LIN {X 0,Y 266.137,Z 368.245,A -85,B 0,C 180,E1 -18633.74,E2 -18633.74} C_VEL
LIN {X 0,Y 268.188,Z 298.553,A -85,B 0,C 180,E1 -18635.636,E2 -18635.636} C_VEL
LIN {X 0,Y 265.756,Z 283.808,A -85,B 0,C 180,E1 -18636.272,E2 -18636.272} C_VEL
LIN {X 0,Y 257.715,Z 261.033,A -85,B 0,C 180,E1 -18637.734,E2 -18637.734} C_VEL
LIN {X 0,Y 256.638,Z 256.402,A -85,B 0,C 180,E1 -18639.459,E2 -18639.459} C_VEL
LIN {X 0,Y 256.319,Z 255.078,A -85,B 0,C 180,E1 -18640.158,E2 -18640.158} C_VEL
LIN {X 0,Y 256.217,Z 255.067,A -85,B 0,C 180,E1 -18644.295,E2 -18644.295} C_VEL
LIN {X 0,Y 256.169,Z 255.06,A -85,B 0,C 180,E1 -18647.567,E2 -18647.567} C_VEL
LIN {X 0,Y 256.112,Z 255.08,A -85,B 0,C 180,E1 -18651.116,E2 -18651.116} C_VEL
LIN {X 0,Y 256.058,Z 255.088,A -85,B 0,C 180,E1 -18655.095,E2 -18655.095} C_VEL
LIN {X 0,Y 256.055,Z 255.092,A -85,B 0,C 180,E1 -18658.578,E2 -18658.578} C_VEL
LIN {X 0,Y 256.047,Z 255.086,A -85,B 0,C 180,E1 -18661.707,E2 -18661.707} C_VEL
LIN {X 0,Y 256.054,Z 255.088,A -85,B 0,C 180,E1 -18665.2,E2 -18665.2} C_VEL
LIN {X 0,Y 256.042,Z 255.078,A -85,B 0,C 180,E1 -18669.15,E2 -18669.15} C_VEL
LIN {X 0,Y 256.002,Z 255.095,A -85,B 0,C 180,E1 -18673.343,E2 -18673.343} C_VEL
LIN {X 0,Y 256.017,Z 255.082,A -85,B 0,C 180,E1 -18677.836,E2 -18677.836} C_VEL
LIN {X 0,Y 256.05,Z 255.079,A -85,B 0,C 180,E1 -18680.864,E2 -18680.864} C_VEL
LIN {X 0,Y 256.067,Z 255.089,A -85,B 0,C 180,E1 -18684.814,E2 -18684.814} C_VEL
LIN {X 0,Y 256.067,Z 255.075,A -85,B 0,C 180,E1 -18688.577,E2 -18688.577} C_VEL
LIN {X 0,Y 256.069,Z 255.074,A -85,B 0,C 180,E1 -18692.196,E2 -18692.196} C_VEL
LIN {X 0,Y 256.079,Z 255.087,A -85,B 0,C 180,E1 -18695.698,E2 -18695.698} C_VEL
LIN {X 0,Y 256.118,Z 255.079,A -85,B 0,C 180,E1 -18699.108,E2 -18699.108} C_VEL
LIN {X 0,Y 256.23,Z 255.045,A -85,B 0,C 180,E1 -18704.088,E2 -18704.088} C_VEL
LIN {X 0,Y 256.288,Z 255.053,A -85,B 0,C 180,E1 -18707.334,E2 -18707.334} C_VEL
LIN {X 0,Y 256.438,Z 255.039,A -85,B 0,C 180,E1 -18710.629,E2 -18710.629} C_VEL
LIN {X 0,Y 256.458,Z 255.029,A -85,B 0,C 180,E1 -18713.713,E2 -18713.713} C_VEL
LIN {X 0,Y 256.703,Z 254.992,A -85,B 0,C 180,E1 -18718.437,E2 -18718.437} C_VEL
LIN {X 0,Y 256.706,Z 255.004,A -85,B 0,C 180,E1 -18721.575,E2 -18721.575} C_VEL
LIN {X 0,Y 256.333,Z 255.048,A -85,B 0,C 180,E1 -18725.241,E2 -18725.241} C_VEL
LIN {X 0,Y 256.073,Z 255.082,A -85,B 0,C 180,E1 -18726.119,E2 -18726.119} C_VEL
LIN {X 0,Y 254.757,Z 255.238,A -85,B 0,C 180,E1 -18727.415,E2 -18727.415} C_VEL
LIN {X 0,Y 250.37,Z 255.78,A -85,B 0,C 180,E1 -18730.434,E2 -18730.434} C_VEL
LIN {X 0,Y 249.286,Z 255.921,A -85,B 0,C 180,E1 -18731.786,E2 -18731.786} C_VEL
LIN {X 0,Y 249.193,Z 255.934,A -85,B 0,C 180,E1 -18732.245,E2 -18732.245} C_VEL
LIN {X 0,Y 249.189,Z 255.946,A -85,B 0,C 180,E1 -18736.473,E2 -18736.473} C_VEL
LIN {X 0,Y 249.062,Z 255.947,A -85,B 0,C 180,E1 -18741.526,E2 -18741.526} C_VEL
LIN {X 0,Y 249.102,Z 255.955,A -85,B 0,C 180,E1 -18745.463,E2 -18745.463} C_VEL
LIN {X 0,Y 249.053,Z 255.949,A -85,B 0,C 180,E1 -18748.976,E2 -18748.976} C_VEL
LIN {X 0,Y 249.046,Z 255.96,A -85,B 0,C 180,E1 -18752.429,E2 -18752.429} C_VEL
LIN {X 0,Y 249.03,Z 255.954,A -85,B 0,C 180,E1 -18756.352,E2 -18756.352} C_VEL
LIN {X 0,Y 248.991,Z 255.968,A -85,B 0,C 180,E1 -18760.487,E2 -18760.487} C_VEL
LIN {X 0,Y 248.982,Z 255.97,A -85,B 0,C 180,E1 -18764.891,E2 -18764.891} C_VEL
LIN {X 0,Y 248.999,Z 255.963,A -85,B 0,C 180,E1 -18767.356,E2 -18767.356} C_VEL
LIN {X 0,Y 249.064,Z 255.951,A -85,B 0,C 180,E1 -18772.202,E2 -18772.202} C_VEL
LIN {X 0,Y 249.119,Z 256.035,A -85,B 0,C 180,E1 -18776.259,E2 -18776.259} C_VEL
LIN {X 0,Y 250.073,Z 260.614,A -85,B 0,C 180,E1 -18778.198,E2 -18778.198} C_VEL
LIN {X 0,Y 251.47,Z 267.192,A -85,B 0,C 180,E1 -18780.671,E2 -18780.671} C_VEL
LIN {X 0,Y 257.562,Z 284.54,A -85,B 0,C 180,E1 -18781.846,E2 -18781.846} C_VEL
LIN {X 0,Y 261.408,Z 311.936,A -85,B 0,C 180,E1 -18783.017,E2 -18783.017} C_VEL
LIN {X 0,Y 259.429,Z 375.405,A -85,B 0,C 180,E1 -18784.795,E2 -18784.795} C_VEL
LIN {X 0,Y 258.511,Z 388.458,A -85,B 0,C 180,E1 -18785.45,E2 -18785.45} C_VEL
LIN {X 0,Y 257.412,Z 400.587,A -85,B 0,C 180,E1 -18786.356,E2 -18786.356} C_VEL
LIN {X 0,Y 255.855,Z 412.812,A -85,B 0,C 180,E1 -18787.594,E2 -18787.594} C_VEL
LIN {X 0,Y 254.121,Z 424.423,A -85,B 0,C 180,E1 -18789.138,E2 -18789.138} C_VEL
LIN {X 0,Y 252.687,Z 434.635,A -85,B 0,C 180,E1 -18790.868,E2 -18790.868} C_VEL
LIN {X 0,Y 251.17,Z 444.299,A -85,B 0,C 180,E1 -18792.912,E2 -18792.912} C_VEL
LIN {X 0,Y 249.834,Z 451.998,A -85,B 0,C 180,E1 -18794.915,E2 -18794.915} C_VEL
LIN {X 0,Y 248.539,Z 459.526,A -85,B 0,C 180,E1 -18797.339,E2 -18797.339} C_VEL
LIN {X 0,Y 247.851,Z 464.648,A -85,B 0,C 180,E1 -18799.376,E2 -18799.376} C_VEL
LIN {X 0,Y 247.28,Z 469.596,A -85,B 0,C 180,E1 -18801.828,E2 -18801.828} C_VEL
LIN {X 0,Y 246.932,Z 473.388,A -85,B 0,C 180,E1 -18804.281,E2 -18804.281} C_VEL
LIN {X 0,Y 246.846,Z 476.14,A -85,B 0,C 180,E1 -18806.733,E2 -18806.733} C_VEL
LIN {X 0,Y 246.87,Z 477.431,A -85,B 0,C 180,E1 -18808.366,E2 -18808.366} C_VEL
LIN {X 0,Y 246.902,Z 478.324,A -85,B 0,C 180,E1 -18809.997,E2 -18809.997} C_VEL
LIN {X 0,Y 246.868,Z 478.796,A -85,B 0,C 180,E1 -18811.629,E2 -18811.629} C_VEL
LIN {X 0,Y 246.938,Z 478.529,A -85,B 0,C 180,E1 -18814.895,E2 -18814.895} C_VEL
LIN {X 0,Y 247.416,Z 476.728,A -85,B 0,C 180,E1 -18818.163,E2 -18818.163} C_VEL
LIN {X 0,Y 248.497,Z 473.247,A -85,B 0,C 180,E1 -18821.416,E2 -18821.416} C_VEL
LIN {X 0,Y 249.736,Z 469.498,A -85,B 0,C 180,E1 -18823.837,E2 -18823.837} C_VEL
LIN {X 0,Y 251.418,Z 464.657,A -85,B 0,C 180,E1 -18826.23,E2 -18826.23} C_VEL
LIN {X 0,Y 253.621,Z 458.573,A -85,B 0,C 180,E1 -18828.58,E2 -18828.58} C_VEL
LIN {X 0,Y 255.955,Z 451.054,A -85,B 0,C 180,E1 -18830.91,E2 -18830.91} C_VEL
LIN {X 0,Y 258.334,Z 443.384,A -85,B 0,C 180,E1 -18832.807,E2 -18832.807} C_VEL
LIN {X 0,Y 261.366,Z 432.989,A -85,B 0,C 180,E1 -18834.841,E2 -18834.841} C_VEL
LIN {X 0,Y 264.043,Z 422.455,A -85,B 0,C 180,E1 -18836.474,E2 -18836.474} C_VEL
LIN {X 0,Y 266.396,Z 412.289,A -85,B 0,C 180,E1 -18837.706,E2 -18837.706} C_VEL
LIN {X 0,Y 268.56,Z 400.294,A -85,B 0,C 180,E1 -18838.845,E2 -18838.845} C_VEL
LIN {X 0,Y 270.494,Z 386.734,A -85,B 0,C 180,E1 -18839.761,E2 -18839.761} C_VEL
LIN {X 0,Y 271.818,Z 373.636,A -85,B 0,C 180,E1 -18840.331,E2 -18840.331} C_VEL
LIN {X 0,Y 274.314,Z 316.425,A -85,B 0,C 180,E1 -18841.884,E2 -18841.884} C_VEL
LIN {X 0,Y 272.34,Z 305.437,A -85,B 0,C 180,E1 -18842.588,E2 -18842.588} C_VEL
LIN {X 0,Y 266.065,Z 291.58,A -85,B 0,C 180,E1 -18844.185,E2 -18844.185} C_VEL
LIN {X 0,Y 259.208,Z 278.747,A -85,B 0,C 180,E1 -18845.979,E2 -18845.979} C_VEL
LIN {X 0,Y 254.374,Z 270.391,A -85,B 0,C 180,E1 -18847.317,E2 -18847.317} C_VEL
LIN {X 0,Y 251.997,Z 266.139,A -85,B 0,C 180,E1 -18848.107,E2 -18848.107} C_VEL
LIN {X 0,Y 249.939,Z 259.099,A -85,B 0,C 180,E1 -18851.81,E2 -18851.81} C_VEL
LIN {X 0,Y 249.002,Z 256.02,A -85,B 0,C 180,E1 -18853.712,E2 -18853.712} C_VEL
LIN {X 0,Y 248.984,Z 255.947,A -85,B 0,C 180,E1 -18857.35,E2 -18857.35} C_VEL
LIN {X 0,Y 249.039,Z 255.965,A -85,B 0,C 180,E1 -18862.197,E2 -18862.197} C_VEL
LIN {X 0,Y 249.044,Z 255.964,A -85,B 0,C 180,E1 -18865.633,E2 -18865.633} C_VEL
LIN {X 0,Y 249.002,Z 255.968,A -85,B 0,C 180,E1 -18869.46,E2 -18869.46} C_VEL
LIN {X 0,Y 249.023,Z 255.965,A -85,B 0,C 180,E1 -18873.151,E2 -18873.151} C_VEL
LIN {X 0,Y 249.004,Z 255.969,A -85,B 0,C 180,E1 -18876.719,E2 -18876.719} C_VEL
LIN {X 0,Y 249.053,Z 255.957,A -85,B 0,C 180,E1 -18880.201,E2 -18880.201} C_VEL
LIN {X 0,Y 249.152,Z 255.937,A -85,B 0,C 180,E1 -18883.61,E2 -18883.61} C_VEL
LIN {X 0,Y 249.182,Z 255.935,A -85,B 0,C 180,E1 -18886.954,E2 -18886.954} C_VEL
LIN {X 0,Y 249.375,Z 255.922,A -85,B 0,C 180,E1 -18890.516,E2 -18890.516} C_VEL
LIN {X 0,Y 249.418,Z 255.907,A -85,B 0,C 180,E1 -18893.522,E2 -18893.522} C_VEL
LIN {X 0,Y 249.645,Z 255.885,A -85,B 0,C 180,E1 -18898.381,E2 -18898.381} C_VEL
LIN {X 0,Y 249.643,Z 255.877,A -85,B 0,C 180,E1 -18901.607,E2 -18901.607} C_VEL
LIN {X 0,Y 249.404,Z 255.911,A -85,B 0,C 180,E1 -18906.541,E2 -18906.541} C_VEL
LIN {X 0,Y 249.325,Z 255.918,A -85,B 0,C 180,E1 -18909.73,E2 -18909.73} C_VEL
LIN {X 0,Y 249.159,Z 255.949,A -85,B 0,C 180,E1 -18914.699,E2 -18914.699} C_VEL
LIN {X 0,Y 249.09,Z 255.958,A -85,B 0,C 180,E1 -18918.074,E2 -18918.074} C_VEL
LIN {X 0,Y 249.058,Z 255.962,A -85,B 0,C 180,E1 -18921.513,E2 -18921.513} C_VEL
LIN {X 0,Y 249.092,Z 255.953,A -85,B 0,C 180,E1 -18925.47,E2 -18925.47} C_VEL
LIN {X 0,Y 249.106,Z 256.1,A -85,B 0,C 180,E1 -18927.735,E2 -18927.735} C_VEL
LIN {X 0,Y 250.653,Z 261.397,A -85,B 0,C 180,E1 -18930.652,E2 -18930.652} C_VEL
LIN {X 0,Y 253.349,Z 265.798,A -85,B 0,C 180,E1 -18931.507,E2 -18931.507} C_VEL
LIN {X 0,Y 259.971,Z 276.7,A -85,B 0,C 180,E1 -18933.334,E2 -18933.334} C_VEL
LIN {X 0,Y 266.437,Z 288.519,A -85,B 0,C 180,E1 -18935.01,E2 -18935.01} C_VEL
LIN {X 0,Y 272.648,Z 301.584,A -85,B 0,C 180,E1 -18936.567,E2 -18936.567} C_VEL
LIN {X 0,Y 274.698,Z 306.633,A -85,B 0,C 180,E1 -18937.083,E2 -18937.083} C_VEL
LIN {X 0,Y 271.808,Z 369.159,A -85,B 0,C 180,E1 -18938.781,E2 -18938.781} C_VEL
LIN {X 0,Y 270.473,Z 383.002,A -85,B 0,C 180,E1 -18939.451,E2 -18939.451} C_VEL
LIN {X 0,Y 268.856,Z 394.598,A -85,B 0,C 180,E1 -18940.277,E2 -18940.277} C_VEL
LIN {X 0,Y 266.755,Z 406.217,A -85,B 0,C 180,E1 -18941.393,E2 -18941.393} C_VEL
LIN {X 0,Y 264.379,Z 417.086,A -85,B 0,C 180,E1 -18942.751,E2 -18942.751} C_VEL
LIN {X 0,Y 261.727,Z 427.447,A -85,B 0,C 180,E1 -18944.386,E2 -18944.386} C_VEL
LIN {X 0,Y 259.026,Z 436.754,A -85,B 0,C 180,E1 -18946.225,E2 -18946.225} C_VEL
LIN {X 0,Y 256.323,Z 445.387,A -85,B 0,C 180,E1 -18948.386,E2 -18948.386} C_VEL
LIN {X 0,Y 253.701,Z 453.161,A -85,B 0,C 180,E1 -18950.852,E2 -18950.852} C_VEL
LIN {X 0,Y 251.75,Z 458.782,A -85,B 0,C 180,E1 -18953.119,E2 -18953.119} C_VEL
LIN {X 0,Y 249.937,Z 463.917,A -85,B 0,C 180,E1 -18955.783,E2 -18955.783} C_VEL
LIN {X 0,Y 248.879,Z 466.963,A -85,B 0,C 180,E1 -18957.888,E2 -18957.888} C_VEL
LIN {X 0,Y 248.228,Z 468.67,A -85,B 0,C 180,E1 -18959.364,E2 -18959.364} C_VEL
LIN {X 0,Y 247.464,Z 470.612,A -85,B 0,C 180,E1 -18961.673,E2 -18961.673} C_VEL
LIN {X 0,Y 246.744,Z 471.965,A -85,B 0,C 180,E1 -18964.71,E2 -18964.71} C_VEL
LIN {X 0,Y 246.552,Z 472.109,A -85,B 0,C 180,E1 -18966.483,E2 -18966.483} C_VEL
LIN {X 0,Y 246.455,Z 471.786,A -85,B 0,C 180,E1 -18968.243,E2 -18968.243} C_VEL
LIN {X 0,Y 246.454,Z 470.925,A -85,B 0,C 180,E1 -18970.202,E2 -18970.202} C_VEL
LIN {X 0,Y 246.534,Z 469.817,A -85,B 0,C 180,E1 -18971.728,E2 -18971.728} C_VEL
LIN {X 0,Y 246.834,Z 467.127,A -85,B 0,C 180,E1 -18974.309,E2 -18974.309} C_VEL
LIN {X 0,Y 247.376,Z 463.344,A -85,B 0,C 180,E1 -18976.866,E2 -18976.866} C_VEL
LIN {X 0,Y 248.02,Z 458.394,A -85,B 0,C 180,E1 -18979.389,E2 -18979.389} C_VEL
LIN {X 0,Y 248.928,Z 452.128,A -85,B 0,C 180,E1 -18981.887,E2 -18981.887} C_VEL
LIN {X 0,Y 250.258,Z 444.298,A -85,B 0,C 180,E1 -18984.362,E2 -18984.362} C_VEL
LIN {X 0,Y 251.601,Z 436.25,A -85,B 0,C 180,E1 -18986.399,E2 -18986.399} C_VEL
LIN {X 0,Y 253.197,Z 426.392,A -85,B 0,C 180,E1 -18988.412,E2 -18988.412} C_VEL
LIN {X 0,Y 254.93,Z 415.392,A -85,B 0,C 180,E1 -18990.2,E2 -18990.2} C_VEL
LIN {X 0,Y 256.331,Z 404.71,A -85,B 0,C 180,E1 -18991.574,E2 -18991.574} C_VEL
LIN {X 0,Y 257.753,Z 391.808,A -85,B 0,C 180,E1 -18992.835,E2 -18992.835} C_VEL
LIN {X 0,Y 258.851,Z 378.874,A -85,B 0,C 180,E1 -18993.748,E2 -18993.748} C_VEL
LIN {X 0,Y 259.553,Z 366.329,A -85,B 0,C 180,E1 -18994.321,E2 -18994.321} C_VEL
LIN {X 0,Y 261.524,Z 298.925,A -85,B 0,C 180,E1 -18996.192,E2 -18996.192} C_VEL
LIN {X 0,Y 259.301,Z 285.865,A -85,B 0,C 180,E1 -18996.782,E2 -18996.782} C_VEL
LIN {X 0,Y 251.041,Z 262.781,A -85,B 0,C 180,E1 -18998.286,E2 -18998.286} C_VEL
LIN {X 0,Y 250.4,Z 260.74,A -85,B 0,C 180,E1 -18998.525,E2 -18998.525} C_VEL
LIN {X 0,Y 249.255,Z 255.976,A -85,B 0,C 180,E1 -19000.562,E2 -19000.562} C_VEL
LIN {X 0,Y 249.164,Z 255.94,A -85,B 0,C 180,E1 -19004.708,E2 -19004.708} C_VEL
LIN {X 0,Y 249.099,Z 255.945,A -85,B 0,C 180,E1 -19008.083,E2 -19008.083} C_VEL
LIN {X 0,Y 249.049,Z 255.958,A -85,B 0,C 180,E1 -19011.524,E2 -19011.524} C_VEL
LIN {X 0,Y 249.019,Z 255.966,A -85,B 0,C 180,E1 -19015.447,E2 -19015.447} C_VEL
LIN {X 0,Y 249.003,Z 255.969,A -85,B 0,C 180,E1 -19018.977,E2 -19018.977} C_VEL
LIN {X 0,Y 249.002,Z 255.959,A -85,B 0,C 180,E1 -19022.433,E2 -19022.433} C_VEL
LIN {X 0,Y 248.989,Z 255.972,A -85,B 0,C 180,E1 -19026.355,E2 -19026.355} C_VEL
LIN {X 0,Y 248.957,Z 255.96,A -85,B 0,C 180,E1 -19030.49,E2 -19030.49} C_VEL
LIN {X 0,Y 248.943,Z 255.975,A -85,B 0,C 180,E1 -19034.896,E2 -19034.896} C_VEL
LIN {X 0,Y 248.962,Z 255.961,A -85,B 0,C 180,E1 -19037.362,E2 -19037.362} C_VEL
LIN {X 0,Y 249.021,Z 255.96,A -85,B 0,C 180,E1 -19042.211,E2 -19042.211} C_VEL
LIN {X 0,Y 249.031,Z 255.961,A -85,B 0,C 180,E1 -19045.647,E2 -19045.647} C_VEL
LIN {X 0,Y 248.984,Z 255.946,A -85,B 0,C 180,E1 -19049.473,E2 -19049.473} C_VEL
LIN {X 0,Y 249.002,Z 255.957,A -85,B 0,C 180,E1 -19053.162,E2 -19053.162} C_VEL
LIN {X 0,Y 249.001,Z 255.967,A -85,B 0,C 180,E1 -19056.733,E2 -19056.733} C_VEL
LIN {X 0,Y 249.054,Z 255.949,A -85,B 0,C 180,E1 -19060.214,E2 -19060.214} C_VEL
LIN {X 0,Y 249.158,Z 255.921,A -85,B 0,C 180,E1 -19063.623,E2 -19063.623} C_VEL
LIN {X 0,Y 249.212,Z 255.933,A -85,B 0,C 180,E1 -19066.968,E2 -19066.968} C_VEL
LIN {X 0,Y 249.388,Z 255.918,A -85,B 0,C 180,E1 -19070.529,E2 -19070.529} C_VEL
LIN {X 0,Y 249.43,Z 255.906,A -85,B 0,C 180,E1 -19073.535,E2 -19073.535} C_VEL
LIN {X 0,Y 249.664,Z 255.866,A -85,B 0,C 180,E1 -19078.393,E2 -19078.393} C_VEL
LIN {X 0,Y 249.666,Z 255.881,A -85,B 0,C 180,E1 -19081.619,E2 -19081.619} C_VEL
LIN {X 0,Y 249.431,Z 255.905,A -85,B 0,C 180,E1 -19086.477,E2 -19086.477} C_VEL
LIN {X 0,Y 249.345,Z 255.898,A -85,B 0,C 180,E1 -19089.742,E2 -19089.742} C_VEL
LIN {X 0,Y 249.193,Z 255.934,A -85,B 0,C 180,E1 -19092.245,E2 -19092.245} C_VEL
LIN {X 0,Y 248.505,Z 256.027,A -85,B 0,C 180,E1 -19093.595,E2 -19093.595} C_VEL
LIN {X 0,Y 245.616,Z 256.388,A -85,B 0,C 180,E1 -19095.794,E2 -19095.794} C_VEL
LIN {X 0,Y 243.16,Z 256.689,A -85,B 0,C 180,E1 -19097.586,E2 -19097.586} C_VEL
LIN {X 0,Y 242.094,Z 256.814,A -85,B 0,C 180,E1 -19098.976,E2 -19098.976} C_VEL
LIN {X 0,Y 242.001,Z 256.821,A -85,B 0,C 180,E1 -19099.448,E2 -19099.448} C_VEL
LIN {X 0,Y 242.04,Z 256.832,A -85,B 0,C 180,E1 -19103.992,E2 -19103.992} C_VEL
LIN {X 0,Y 241.984,Z 256.834,A -85,B 0,C 180,E1 -19107.696,E2 -19107.696} C_VEL
LIN {X 0,Y 241.971,Z 256.839,A -85,B 0,C 180,E1 -19111.527,E2 -19111.527} C_VEL
LIN {X 0,Y 241.998,Z 256.832,A -85,B 0,C 180,E1 -19115.59,E2 -19115.59} C_VEL
LIN {X 0,Y 241.949,Z 256.848,A -85,B 0,C 180,E1 -19119.727,E2 -19119.727} C_VEL
LIN {X 0,Y 241.917,Z 256.85,A -85,B 0,C 180,E1 -19124.212,E2 -19124.212} C_VEL
LIN {X 0,Y 241.928,Z 256.846,A -85,B 0,C 180,E1 -19128.073,E2 -19128.073} C_VEL
LIN {X 0,Y 242.004,Z 256.83,A -85,B 0,C 180,E1 -19132.418,E2 -19132.418} C_VEL
LIN {X 0,Y 242.061,Z 256.904,A -85,B 0,C 180,E1 -19135.766,E2 -19135.766} C_VEL
LIN {X 0,Y 243.466,Z 263.76,A -85,B 0,C 180,E1 -19138.692,E2 -19138.692} C_VEL
LIN {X 0,Y 244.276,Z 267.244,A -85,B 0,C 180,E1 -19139.961,E2 -19139.961} C_VEL
LIN {X 0,Y 250.79,Z 285.555,A -85,B 0,C 180,E1 -19141.238,E2 -19141.238} C_VEL
LIN {X 0,Y 251.532,Z 289.12,A -85,B 0,C 180,E1 -19141.422,E2 -19141.422} C_VEL
LIN {X 0,Y 254.74,Z 313.439,A -85,B 0,C 180,E1 -19142.477,E2 -19142.477} C_VEL
LIN {X 0,Y 252.762,Z 374.998,A -85,B 0,C 180,E1 -19144.247,E2 -19144.247} C_VEL
LIN {X 0,Y 251.837,Z 388.159,A -85,B 0,C 180,E1 -19144.92,E2 -19144.92} C_VEL
LIN {X 0,Y 250.626,Z 400.901,A -85,B 0,C 180,E1 -19145.896,E2 -19145.896} C_VEL
LIN {X 0,Y 249.027,Z 413.005,A -85,B 0,C 180,E1 -19147.164,E2 -19147.164} C_VEL
LIN {X 0,Y 247.246,Z 424.563,A -85,B 0,C 180,E1 -19148.749,E2 -19148.749} C_VEL
LIN {X 0,Y 245.833,Z 434.191,A -85,B 0,C 180,E1 -19150.421,E2 -19150.421} C_VEL
LIN {X 0,Y 244.362,Z 443.525,A -85,B 0,C 180,E1 -19152.421,E2 -19152.421} C_VEL
LIN {X 0,Y 242.956,Z 451.342,A -85,B 0,C 180,E1 -19154.477,E2 -19154.477} C_VEL
LIN {X 0,Y 241.575,Z 458.967,A -85,B 0,C 180,E1 -19156.967,E2 -19156.967} C_VEL
LIN {X 0,Y 240.852,Z 464.178,A -85,B 0,C 180,E1 -19159.064,E2 -19159.064} C_VEL
LIN {X 0,Y 240.226,Z 469.205,A -85,B 0,C 180,E1 -19161.586,E2 -19161.586} C_VEL
LIN {X 0,Y 239.851,Z 473.071,A -85,B 0,C 180,E1 -19164.111,E2 -19164.111} C_VEL
LIN {X 0,Y 239.755,Z 475.893,A -85,B 0,C 180,E1 -19166.636,E2 -19166.636} C_VEL
LIN {X 0,Y 239.784,Z 477.218,A -85,B 0,C 180,E1 -19168.318,E2 -19168.318} C_VEL
LIN {X 0,Y 239.814,Z 478.144,A -85,B 0,C 180,E1 -19169.997,E2 -19169.997} C_VEL
LIN {X 0,Y 239.782,Z 478.672,A -85,B 0,C 180,E1 -19171.677,E2 -19171.677} C_VEL
LIN {X 0,Y 239.857,Z 478.478,A -85,B 0,C 180,E1 -19175.04,E2 -19175.04} C_VEL
LIN {X 0,Y 240.39,Z 476.757,A -85,B 0,C 180,E1 -19178.403,E2 -19178.403} C_VEL
LIN {X 0,Y 240.879,Z 475.272,A -85,B 0,C 180,E1 -19180.079,E2 -19180.079} C_VEL
LIN {X 0,Y 241.905,Z 472.275,A -85,B 0,C 180,E1 -19182.583,E2 -19182.583} C_VEL
LIN {X 0,Y 243.331,Z 468.251,A -85,B 0,C 180,E1 -19185.064,E2 -19185.064} C_VEL
LIN {X 0,Y 245.701,Z 462.088,A -85,B 0,C 180,E1 -19187.905,E2 -19187.905} C_VEL
LIN {X 0,Y 248.18,Z 455.4,A -85,B 0,C 180,E1 -19190.295,E2 -19190.295} C_VEL
LIN {X 0,Y 250.244,Z 448.919,A -85,B 0,C 180,E1 -19192.191,E2 -19192.191} C_VEL
LIN {X 0,Y 252.968,Z 440.475,A -85,B 0,C 180,E1 -19194.189,E2 -19194.189} C_VEL
LIN {X 0,Y 255.876,Z 430.571,A -85,B 0,C 180,E1 -19196.067,E2 -19196.067} C_VEL
LIN {X 0,Y 258.717,Z 419.428,A -85,B 0,C 180,E1 -19197.72,E2 -19197.72} C_VEL
LIN {X 0,Y 261.192,Z 408.542,A -85,B 0,C 180,E1 -19198.966,E2 -19198.966} C_VEL
LIN {X 0,Y 263.381,Z 396.551,A -85,B 0,C 180,E1 -19200.018,E2 -19200.018} C_VEL
LIN {X 0,Y 265.106,Z 384.122,A -85,B 0,C 180,E1 -19200.796,E2 -19200.796} C_VEL
LIN {X 0,Y 266.375,Z 370.258,A -85,B 0,C 180,E1 -19201.338,E2 -19201.338} C_VEL
LIN {X 0,Y 268.649,Z 317.236,A -85,B 0,C 180,E1 -19202.81,E2 -19202.81} C_VEL
LIN {X 0,Y 267.016,Z 308.276,A -85,B 0,C 180,E1 -19203.414,E2 -19203.414} C_VEL
LIN {X 0,Y 261.056,Z 295.118,A -85,B 0,C 180,E1 -19204.998,E2 -19204.998} C_VEL
LIN {X 0,Y 254.404,Z 282.5,A -85,B 0,C 180,E1 -19206.828,E2 -19206.828} C_VEL
LIN {X 0,Y 250.213,Z 275.207,A -85,B 0,C 180,E1 -19208.053,E2 -19208.053} C_VEL
LIN {X 0,Y 247.079,Z 270.154,A -85,B 0,C 180,E1 -19209.001,E2 -19209.001} C_VEL
LIN {X 0,Y 244.693,Z 266.008,A -85,B 0,C 180,E1 -19209.849,E2 -19209.849} C_VEL
LIN {X 0,Y 242.702,Z 259.318,A -85,B 0,C 180,E1 -19213.613,E2 -19213.613} C_VEL
LIN {X 0,Y 241.927,Z 256.881,A -85,B 0,C 180,E1 -19215.286,E2 -19215.286} C_VEL
LIN {X 0,Y 241.908,Z 256.851,A -85,B 0,C 180,E1 -19219.052,E2 -19219.052} C_VEL
LIN {X 0,Y 241.982,Z 256.844,A -85,B 0,C 180,E1 -19222.41,E2 -19222.41} C_VEL
LIN {X 0,Y 241.98,Z 256.836,A -85,B 0,C 180,E1 -19226.501,E2 -19226.501} C_VEL
LIN {X 0,Y 241.976,Z 256.834,A -85,B 0,C 180,E1 -19230.607,E2 -19230.607} C_VEL
LIN {X 0,Y 241.995,Z 256.832,A -85,B 0,C 180,E1 -19234.191,E2 -19234.191} C_VEL
LIN {X 0,Y 241.982,Z 256.832,A -85,B 0,C 180,E1 -19238.332,E2 -19238.332} C_VEL
LIN {X 0,Y 242.108,Z 256.814,A -85,B 0,C 180,E1 -19243.312,E2 -19243.312} C_VEL
LIN {X 0,Y 242.159,Z 256.807,A -85,B 0,C 180,E1 -19248.272,E2 -19248.272} C_VEL
LIN {X 0,Y 242.364,Z 256.783,A -85,B 0,C 180,E1 -19251.657,E2 -19251.657} C_VEL
LIN {X 0,Y 242.388,Z 256.781,A -85,B 0,C 180,E1 -19253.334,E2 -19253.334} C_VEL
LIN {X 0,Y 242.604,Z 256.761,A -85,B 0,C 180,E1 -19258.334,E2 -19258.334} C_VEL
LIN {X 0,Y 242.603,Z 256.753,A -85,B 0,C 180,E1 -19261.654,E2 -19261.654} C_VEL
LIN {X 0,Y 242.379,Z 256.787,A -85,B 0,C 180,E1 -19266.654,E2 -19266.654} C_VEL
LIN {X 0,Y 242.248,Z 256.8,A -85,B 0,C 180,E1 -19270.018,E2 -19270.018} C_VEL
LIN {X 0,Y 242.116,Z 256.827,A -85,B 0,C 180,E1 -19275.137,E2 -19275.137} C_VEL
LIN {X 0,Y 242.028,Z 256.837,A -85,B 0,C 180,E1 -19278.62,E2 -19278.62} C_VEL
LIN {X 0,Y 241.982,Z 256.838,A -85,B 0,C 180,E1 -19282.175,E2 -19282.175} C_VEL
LIN {X 0,Y 242.054,Z 257.006,A -85,B 0,C 180,E1 -19286.226,E2 -19286.226} C_VEL
LIN {X 0,Y 243.379,Z 261.453,A -85,B 0,C 180,E1 -19288.859,E2 -19288.859} C_VEL
LIN {X 0,Y 246.017,Z 265.751,A -85,B 0,C 180,E1 -19289.79,E2 -19289.79} C_VEL
LIN {X 0,Y 252.809,Z 276.425,A -85,B 0,C 180,E1 -19291.816,E2 -19291.816} C_VEL
LIN {X 0,Y 259.725,Z 288.718,A -85,B 0,C 180,E1 -19293.741,E2 -19293.741} C_VEL
LIN {X 0,Y 266.785,Z 303.208,A -85,B 0,C 180,E1 -19295.6,E2 -19295.6} C_VEL
LIN {X 0,Y 269.114,Z 309.085,A -85,B 0,C 180,E1 -19296.22,E2 -19296.22} C_VEL
LIN {X 0,Y 266.189,Z 368.862,A -85,B 0,C 180,E1 -19297.857,E2 -19297.857} C_VEL
LIN {X 0,Y 264.872,Z 382.098,A -85,B 0,C 180,E1 -19298.492,E2 -19298.492} C_VEL
LIN {X 0,Y 263.012,Z 394.921,A -85,B 0,C 180,E1 -19299.407,E2 -19299.407} C_VEL
LIN {X 0,Y 260.643,Z 407.357,A -85,B 0,C 180,E1 -19300.647,E2 -19300.647} C_VEL
LIN {X 0,Y 258.057,Z 418.451,A -85,B 0,C 180,E1 -19302.091,E2 -19302.091} C_VEL
LIN {X 0,Y 255.484,Z 427.937,A -85,B 0,C 180,E1 -19303.644,E2 -19303.644} C_VEL
LIN {X 0,Y 252.812,Z 436.717,A -85,B 0,C 180,E1 -19305.422,E2 -19305.422} C_VEL
LIN {X 0,Y 249.996,Z 445.212,A -85,B 0,C 180,E1 -19307.573,E2 -19307.573} C_VEL
LIN {X 0,Y 247.189,Z 453.138,A -85,B 0,C 180,E1 -19310.131,E2 -19310.131} C_VEL
LIN {X 0,Y 244.761,Z 459.789,A -85,B 0,C 180,E1 -19312.919,E2 -19312.919} C_VEL
LIN {X 0,Y 242.884,Z 464.666,A -85,B 0,C 180,E1 -19315.654,E2 -19315.654} C_VEL
LIN {X 0,Y 241.516,Z 468.249,A -85,B 0,C 180,E1 -19318.416,E2 -19318.416} C_VEL
LIN {X 0,Y 240.472,Z 470.683,A -85,B 0,C 180,E1 -19321.238,E2 -19321.238} C_VEL
LIN {X 0,Y 239.784,Z 471.931,A -85,B 0,C 180,E1 -19323.922,E2 -19323.922} C_VEL
LIN {X 0,Y 239.54,Z 472.218,A -85,B 0,C 180,E1 -19325.751,E2 -19325.751} C_VEL
LIN {X 0,Y 239.366,Z 472.028,A -85,B 0,C 180,E1 -19327.565,E2 -19327.565} C_VEL
LIN {X 0,Y 239.353,Z 471.084,A -85,B 0,C 180,E1 -19329.959,E2 -19329.959} C_VEL
LIN {X 0,Y 239.551,Z 468.732,A -85,B 0,C 180,E1 -19332.942,E2 -19332.942} C_VEL
LIN {X 0,Y 239.897,Z 466.13,A -85,B 0,C 180,E1 -19335.153,E2 -19335.153} C_VEL
LIN {X 0,Y 240.375,Z 462.741,A -85,B 0,C 180,E1 -19337.336,E2 -19337.336} C_VEL
LIN {X 0,Y 241.087,Z 457.605,A -85,B 0,C 180,E1 -19339.929,E2 -19339.929} C_VEL
LIN {X 0,Y 242.109,Z 451.126,A -85,B 0,C 180,E1 -19342.497,E2 -19342.497} C_VEL
LIN {X 0,Y 243.459,Z 442.974,A -85,B 0,C 180,E1 -19345.034,E2 -19345.034} C_VEL
LIN {X 0,Y 244.88,Z 434.637,A -85,B 0,C 180,E1 -19347.124,E2 -19347.124} C_VEL
LIN {X 0,Y 246.475,Z 425.423,A -85,B 0,C 180,E1 -19348.999,E2 -19348.999} C_VEL
LIN {X 0,Y 248.077,Z 415.635,A -85,B 0,C 180,E1 -19350.611,E2 -19350.611} C_VEL
LIN {X 0,Y 249.515,Z 405.005,A -85,B 0,C 180,E1 -19352.02,E2 -19352.02} C_VEL
LIN {X 0,Y 250.891,Z 393.294,A -85,B 0,C 180,E1 -19353.214,E2 -19353.214} C_VEL
LIN {X 0,Y 252.088,Z 380.07,A -85,B 0,C 180,E1 -19354.199,E2 -19354.199} C_VEL
LIN {X 0,Y 252.845,Z 367.253,A -85,B 0,C 180,E1 -19354.83,E2 -19354.83} C_VEL
LIN {X 0,Y 254.898,Z 299.64,A -85,B 0,C 180,E1 -19356.765,E2 -19356.765} C_VEL
LIN {X 0,Y 252.904,Z 287.906,A -85,B 0,C 180,E1 -19357.315,E2 -19357.315} C_VEL
LIN {X 0,Y 245.05,Z 265.909,A -85,B 0,C 180,E1 -19358.798,E2 -19358.798} C_VEL
LIN {X 0,Y 243.205,Z 261.105,A -85,B 0,C 180,E1 -19359.203,E2 -19359.203} C_VEL
LIN {X 0,Y 242.208,Z 256.922,A -85,B 0,C 180,E1 -19360.979,E2 -19360.979} C_VEL
LIN {X 0,Y 242.118,Z 256.809,A -85,B 0,C 180,E1 -19365.146,E2 -19365.146} C_VEL
LIN {X 0,Y 242.034,Z 256.832,A -85,B 0,C 180,E1 -19368.63,E2 -19368.63} C_VEL
LIN {X 0,Y 241.961,Z 256.841,A -85,B 0,C 180,E1 -19372.188,E2 -19372.188} C_VEL
LIN {X 0,Y 241.959,Z 256.841,A -85,B 0,C 180,E1 -19375.832,E2 -19375.832} C_VEL
LIN {X 0,Y 241.94,Z 256.85,A -85,B 0,C 180,E1 -19379.595,E2 -19379.595} C_VEL
LIN {X 0,Y 241.954,Z 256.837,A -85,B 0,C 180,E1 -19383.499,E2 -19383.499} C_VEL
LIN {X 0,Y 241.961,Z 256.842,A -85,B 0,C 180,E1 -19387.59,E2 -19387.59} C_VEL
LIN {X 0,Y 241.887,Z 256.847,A -85,B 0,C 180,E1 -19391.936,E2 -19391.936} C_VEL
LIN {X 0,Y 241.882,Z 256.848,A -85,B 0,C 180,E1 -19396.587,E2 -19396.587} C_VEL
LIN {X 0,Y 241.975,Z 256.837,A -85,B 0,C 180,E1 -19401.65,E2 -19401.65} C_VEL
LIN {X 0,Y 241.965,Z 256.844,A -85,B 0,C 180,E1 -19404.495,E2 -19404.495} C_VEL
LIN {X 0,Y 241.938,Z 256.832,A -85,B 0,C 180,E1 -19408.484,E2 -19408.484} C_VEL
LIN {X 0,Y 241.942,Z 256.832,A -85,B 0,C 180,E1 -19412.313,E2 -19412.313} C_VEL
LIN {X 0,Y 241.974,Z 256.842,A -85,B 0,C 180,E1 -19416.015,E2 -19416.015} C_VEL
LIN {X 0,Y 241.988,Z 256.832,A -85,B 0,C 180,E1 -19419.611,E2 -19419.611} C_VEL
LIN {X 0,Y 242.114,Z 256.796,A -85,B 0,C 180,E1 -19423.325,E2 -19423.325} C_VEL
LIN {X 0,Y 242.179,Z 256.816,A -85,B 0,C 180,E1 -19428.286,E2 -19428.286} C_VEL
LIN {X 0,Y 242.376,Z 256.792,A -85,B 0,C 180,E1 -19431.671,E2 -19431.671} C_VEL
LIN {X 0,Y 242.401,Z 256.783,A -85,B 0,C 180,E1 -19433.347,E2 -19433.347} C_VEL
LIN {X 0,Y 242.624,Z 256.74,A -85,B 0,C 180,E1 -19438.347,E2 -19438.347} C_VEL
LIN {X 0,Y 242.626,Z 256.758,A -85,B 0,C 180,E1 -19441.666,E2 -19441.666} C_VEL
LIN {X 0,Y 242.401,Z 256.779,A -85,B 0,C 180,E1 -19446.666,E2 -19446.666} C_VEL
LIN {X 0,Y 242.274,Z 256.778,A -85,B 0,C 180,E1 -19450.03,E2 -19450.03} C_VEL
LIN {X 0,Y 242.142,Z 256.822,A -85,B 0,C 180,E1 -19455.148,E2 -19455.148} C_VEL
LIN {X 0,Y 242.001,Z 256.821,A -85,B 0,C 180,E1 -19459.448,E2 -19459.448} C_VEL
LIN {X 0,Y 241.332,Z 256.905,A -85,B 0,C 180,E1 -19460.836,E2 -19460.836} C_VEL
LIN {X 0,Y 238.536,Z 257.27,A -85,B 0,C 180,E1 -19463.102,E2 -19463.102} C_VEL
LIN {X 0,Y 235.31,Z 257.68,A -85,B 0,C 180,E1 -19465.896,E2 -19465.896} C_VEL
LIN {X 0,Y 234.946,Z 257.716,A -85,B 0,C 180,E1 -19466.863,E2 -19466.863} C_VEL
LIN {X 0,Y 234.917,Z 257.709,A -85,B 0,C 180,E1 -19470.576,E2 -19470.576} C_VEL
LIN {X 0,Y 234.942,Z 257.718,A -85,B 0,C 180,E1 -19474.643,E2 -19474.643} C_VEL
LIN {X 0,Y 234.932,Z 257.718,A -85,B 0,C 180,E1 -19478.938,E2 -19478.938} C_VEL
LIN {X 0,Y 234.883,Z 257.726,A -85,B 0,C 180,E1 -19484.098,E2 -19484.098} C_VEL
LIN {X 0,Y 234.874,Z 257.727,A -85,B 0,C 180,E1 -19488.827,E2 -19488.827} C_VEL
LIN {X 0,Y 234.939,Z 257.71,A -85,B 0,C 180,E1 -19491.08,E2 -19491.08} C_VEL
LIN {X 0,Y 234.997,Z 257.78,A -85,B 0,C 180,E1 -19495.244,E2 -19495.244} C_VEL
LIN {X 0,Y 236.363,Z 264.217,A -85,B 0,C 180,E1 -19498.103,E2 -19498.103} C_VEL
LIN {X 0,Y 236.97,Z 267.079,A -85,B 0,C 180,E1 -19499.166,E2 -19499.166} C_VEL
LIN {X 0,Y 242.009,Z 280.596,A -85,B 0,C 180,E1 -19500.213,E2 -19500.213} C_VEL
LIN {X 0,Y 244.93,Z 289.669,A -85,B 0,C 180,E1 -19500.802,E2 -19500.802} C_VEL
LIN {X 0,Y 248.154,Z 313.429,A -85,B 0,C 180,E1 -19501.873,E2 -19501.873} C_VEL
LIN {X 0,Y 246.08,Z 375.738,A -85,B 0,C 180,E1 -19503.723,E2 -19503.723} C_VEL
LIN {X 0,Y 245.039,Z 389.377,A -85,B 0,C 180,E1 -19504.459,E2 -19504.459} C_VEL
LIN {X 0,Y 243.748,Z 402.241,A -85,B 0,C 180,E1 -19505.511,E2 -19505.511} C_VEL
LIN {X 0,Y 241.967,Z 414.79,A -85,B 0,C 180,E1 -19506.911,E2 -19506.911} C_VEL
LIN {X 0,Y 240.188,Z 426.005,A -85,B 0,C 180,E1 -19508.543,E2 -19508.543} C_VEL
LIN {X 0,Y 238.557,Z 436.592,A -85,B 0,C 180,E1 -19510.529,E2 -19510.529} C_VEL
LIN {X 0,Y 236.882,Z 446.049,A -85,B 0,C 180,E1 -19512.739,E2 -19512.739} C_VEL
LIN {X 0,Y 235.549,Z 453.425,A -85,B 0,C 180,E1 -19514.864,E2 -19514.864} C_VEL
LIN {X 0,Y 234.294,Z 460.663,A -85,B 0,C 180,E1 -19517.437,E2 -19517.437} C_VEL
LIN {X 0,Y 233.59,Z 465.539,A -85,B 0,C 180,E1 -19519.597,E2 -19519.597} C_VEL
LIN {X 0,Y 233.021,Z 470.253,A -85,B 0,C 180,E1 -19522.197,E2 -19522.197} C_VEL
LIN {X 0,Y 232.698,Z 474.477,A -85,B 0,C 180,E1 -19525.379,E2 -19525.379} C_VEL
LIN {X 0,Y 232.681,Z 477.004,A -85,B 0,C 180,E1 -19528.266,E2 -19528.266} C_VEL
LIN {X 0,Y 232.729,Z 477.964,A -85,B 0,C 180,E1 -19529.997,E2 -19529.997} C_VEL
LIN {X 0,Y 232.679,Z 478.529,A -85,B 0,C 180,E1 -19531.728,E2 -19531.728} C_VEL
LIN {X 0,Y 232.754,Z 478.54,A -85,B 0,C 180,E1 -19534.788,E2 -19534.788} C_VEL
LIN {X 0,Y 232.998,Z 477.79,A -85,B 0,C 180,E1 -19536.927,E2 -19536.927} C_VEL
LIN {X 0,Y 233.866,Z 475.352,A -85,B 0,C 180,E1 -19540.385,E2 -19540.385} C_VEL
LIN {X 0,Y 234.969,Z 472.411,A -85,B 0,C 180,E1 -19542.96,E2 -19542.96} C_VEL
LIN {X 0,Y 236.467,Z 468.454,A -85,B 0,C 180,E1 -19545.512,E2 -19545.512} C_VEL
LIN {X 0,Y 238.558,Z 463.382,A -85,B 0,C 180,E1 -19548.016,E2 -19548.016} C_VEL
LIN {X 0,Y 241.056,Z 457.036,A -85,B 0,C 180,E1 -19550.476,E2 -19550.476} C_VEL
LIN {X 0,Y 243.698,Z 449.454,A -85,B 0,C 180,E1 -19552.82,E2 -19552.82} C_VEL
LIN {X 0,Y 246.56,Z 441.154,A -85,B 0,C 180,E1 -19554.859,E2 -19554.859} C_VEL
LIN {X 0,Y 249.575,Z 431.424,A -85,B 0,C 180,E1 -19556.776,E2 -19556.776} C_VEL
LIN {X 0,Y 252.538,Z 420.582,A -85,B 0,C 180,E1 -19558.459,E2 -19558.459} C_VEL
LIN {X 0,Y 255.445,Z 408.257,A -85,B 0,C 180,E1 -19559.909,E2 -19559.909} C_VEL
LIN {X 0,Y 257.721,Z 396.214,A -85,B 0,C 180,E1 -19560.975,E2 -19560.975} C_VEL
LIN {X 0,Y 259.503,Z 383.895,A -85,B 0,C 180,E1 -19561.747,E2 -19561.747} C_VEL
LIN {X 0,Y 260.785,Z 370.013,A -85,B 0,C 180,E1 -19562.299,E2 -19562.299} C_VEL
LIN {X 0,Y 263.115,Z 318.415,A -85,B 0,C 180,E1 -19563.753,E2 -19563.753} C_VEL
LIN {X 0,Y 261.817,Z 311.218,A -85,B 0,C 180,E1 -19564.256,E2 -19564.256} C_VEL
LIN {X 0,Y 255.594,Z 297.539,A -85,B 0,C 180,E1 -19565.988,E2 -19565.988} C_VEL
LIN {X 0,Y 248.743,Z 284.525,A -85,B 0,C 180,E1 -19568.006,E2 -19568.006} C_VEL
LIN {X 0,Y 243.485,Z 275.59,A -85,B 0,C 180,E1 -19569.644,E2 -19569.644} C_VEL
LIN {X 0,Y 239.692,Z 269.851,A -85,B 0,C 180,E1 -19570.873,E2 -19570.873} C_VEL
LIN {X 0,Y 237.396,Z 265.88,A -85,B 0,C 180,E1 -19571.765,E2 -19571.765} C_VEL
LIN {X 0,Y 235.623,Z 260.126,A -85,B 0,C 180,E1 -19575.257,E2 -19575.257} C_VEL
LIN {X 0,Y 234.877,Z 257.739,A -85,B 0,C 180,E1 -19577.043,E2 -19577.043} C_VEL
LIN {X 0,Y 234.921,Z 257.716,A -85,B 0,C 180,E1 -19581.073,E2 -19581.073} C_VEL
LIN {X 0,Y 234.926,Z 257.723,A -85,B 0,C 180,E1 -19585.355,E2 -19585.355} C_VEL
LIN {X 0,Y 234.899,Z 257.724,A -85,B 0,C 180,E1 -19589.421,E2 -19589.421} C_VEL
LIN {X 0,Y 234.94,Z 257.713,A -85,B 0,C 180,E1 -19593.814,E2 -19593.814} C_VEL
LIN {X 0,Y 234.936,Z 257.708,A -85,B 0,C 180,E1 -19598.957,E2 -19598.957} C_VEL
LIN {X 0,Y 235.05,Z 257.693,A -85,B 0,C 180,E1 -19603.087,E2 -19603.087} C_VEL
LIN {X 0,Y 235.091,Z 257.687,A -85,B 0,C 180,E1 -19607.915,E2 -19607.915} C_VEL
LIN {X 0,Y 235.303,Z 257.664,A -85,B 0,C 180,E1 -19611.405,E2 -19611.405} C_VEL
LIN {X 0,Y 235.34,Z 257.657,A -85,B 0,C 180,E1 -19613.133,E2 -19613.133} C_VEL
LIN {X 0,Y 235.563,Z 257.636,A -85,B 0,C 180,E1 -19618.284,E2 -19618.284} C_VEL
LIN {X 0,Y 235.562,Z 257.63,A -85,B 0,C 180,E1 -19621.703,E2 -19621.703} C_VEL
LIN {X 0,Y 235.331,Z 257.667,A -85,B 0,C 180,E1 -19626.854,E2 -19626.854} C_VEL
LIN {X 0,Y 235.194,Z 257.68,A -85,B 0,C 180,E1 -19630.321,E2 -19630.321} C_VEL
LIN {X 0,Y 235.06,Z 257.702,A -85,B 0,C 180,E1 -19635.603,E2 -19635.603} C_VEL
LIN {X 0,Y 234.968,Z 257.711,A -85,B 0,C 180,E1 -19639.201,E2 -19639.201} C_VEL
LIN {X 0,Y 234.957,Z 257.718,A -85,B 0,C 180,E1 -19643.808,E2 -19643.808} C_VEL
LIN {X 0,Y 234.978,Z 257.876,A -85,B 0,C 180,E1 -19644.51,E2 -19644.51} C_VEL
LIN {X 0,Y 236.154,Z 261.672,A -85,B 0,C 180,E1 -19646.934,E2 -19646.934} C_VEL
LIN {X 0,Y 240.519,Z 268.425,A -85,B 0,C 180,E1 -19648.518,E2 -19648.518} C_VEL
LIN {X 0,Y 244.408,Z 274.405,A -85,B 0,C 180,E1 -19649.771,E2 -19649.771} C_VEL
LIN {X 0,Y 249.54,Z 282.798,A -85,B 0,C 180,E1 -19651.341,E2 -19651.341} C_VEL
LIN {X 0,Y 255.279,Z 293.211,A -85,B 0,C 180,E1 -19653.016,E2 -19653.016} C_VEL
LIN {X 0,Y 261.874,Z 306.957,A -85,B 0,C 180,E1 -19654.834,E2 -19654.834} C_VEL
LIN {X 0,Y 263.434,Z 310.715,A -85,B 0,C 180,E1 -19655.261,E2 -19655.261} C_VEL
LIN {X 0,Y 261.235,Z 358.548,A -85,B 0,C 180,E1 -19656.596,E2 -19656.596} C_VEL
LIN {X 0,Y 260.204,Z 373.678,A -85,B 0,C 180,E1 -19657.101,E2 -19657.101} C_VEL
LIN {X 0,Y 258.633,Z 386.705,A -85,B 0,C 180,E1 -19657.844,E2 -19657.844} C_VEL
LIN {X 0,Y 256.613,Z 398.741,A -85,B 0,C 180,E1 -19658.819,E2 -19658.819} C_VEL
LIN {X 0,Y 254.407,Z 409.323,A -85,B 0,C 180,E1 -19659.955,E2 -19659.955} C_VEL
LIN {X 0,Y 251.549,Z 420.763,A -85,B 0,C 180,E1 -19661.54,E2 -19661.54} C_VEL
LIN {X 0,Y 248.272,Z 431.754,A -85,B 0,C 180,E1 -19663.503,E2 -19663.503} C_VEL
LIN {X 0,Y 245.127,Z 441.171,A -85,B 0,C 180,E1 -19665.651,E2 -19665.651} C_VEL
LIN {X 0,Y 242.12,Z 449.564,A -85,B 0,C 180,E1 -19668.12,E2 -19668.12} C_VEL
LIN {X 0,Y 239.302,Z 456.809,A -85,B 0,C 180,E1 -19670.848,E2 -19670.848} C_VEL
LIN {X 0,Y 237.053,Z 462.439,A -85,B 0,C 180,E1 -19673.637,E2 -19673.637} C_VEL
LIN {X 0,Y 235.166,Z 467.065,A -85,B 0,C 180,E1 -19676.787,E2 -19676.787} C_VEL
LIN {X 0,Y 234.023,Z 469.659,A -85,B 0,C 180,E1 -19679.304,E2 -19679.304} C_VEL
LIN {X 0,Y 233.382,Z 471.023,A -85,B 0,C 180,E1 -19681.199,E2 -19681.199} C_VEL
LIN {X 0,Y 232.878,Z 471.896,A -85,B 0,C 180,E1 -19683.087,E2 -19683.087} C_VEL
LIN {X 0,Y 232.53,Z 472.281,A -85,B 0,C 180,E1 -19685.035,E2 -19685.035} C_VEL
LIN {X 0,Y 232.313,Z 472.223,A -85,B 0,C 180,E1 -19686.844,E2 -19686.844} C_VEL
LIN {X 0,Y 232.25,Z 471.234,A -85,B 0,C 180,E1 -19689.705,E2 -19689.705} C_VEL
LIN {X 0,Y 232.374,Z 469.29,A -85,B 0,C 180,E1 -19692.399,E2 -19692.399} C_VEL
LIN {X 0,Y 232.77,Z 466.406,A -85,B 0,C 180,E1 -19695.02,E2 -19695.02} C_VEL
LIN {X 0,Y 233.367,Z 462.14,A -85,B 0,C 180,E1 -19697.833,E2 -19697.833} C_VEL
LIN {X 0,Y 234.331,Z 455.749,A -85,B 0,C 180,E1 -19700.943,E2 -19700.943} C_VEL
LIN {X 0,Y 235.469,Z 448.771,A -85,B 0,C 180,E1 -19703.576,E2 -19703.576} C_VEL
LIN {X 0,Y 236.78,Z 441.618,A -85,B 0,C 180,E1 -19705.747,E2 -19705.747} C_VEL
LIN {X 0,Y 238.303,Z 432.991,A -85,B 0,C 180,E1 -19707.89,E2 -19707.89} C_VEL
LIN {X 0,Y 240.201,Z 422.248,A -85,B 0,C 180,E1 -19710.003,E2 -19710.003} C_VEL
LIN {X 0,Y 241.856,Z 411.6,A -85,B 0,C 180,E1 -19711.668,E2 -19711.668} C_VEL
LIN {X 0,Y 243.393,Z 399.888,A -85,B 0,C 180,E1 -19713.106,E2 -19713.106} C_VEL
LIN {X 0,Y 244.739,Z 387.658,A -85,B 0,C 180,E1 -19714.222,E2 -19714.222} C_VEL
LIN {X 0,Y 245.811,Z 374.402,A -85,B 0,C 180,E1 -19715.077,E2 -19715.077} C_VEL
LIN {X 0,Y 246.464,Z 361.726,A -85,B 0,C 180,E1 -19715.576,E2 -19715.576} C_VEL
LIN {X 0,Y 248.334,Z 300.555,A -85,B 0,C 180,E1 -19717.352,E2 -19717.352} C_VEL
LIN {X 0,Y 246.632,Z 290.296,A -85,B 0,C 180,E1 -19717.847,E2 -19717.847} C_VEL
LIN {X 0,Y 238.609,Z 267.788,A -85,B 0,C 180,E1 -19719.411,E2 -19719.411} C_VEL
LIN {X 0,Y 236.029,Z 261.488,A -85,B 0,C 180,E1 -19719.935,E2 -19719.935} C_VEL
LIN {X 0,Y 235.707,Z 260.214,A -85,B 0,C 180,E1 -19720.328,E2 -19720.328} C_VEL
LIN {X 0,Y 235.126,Z 257.754,A -85,B 0,C 180,E1 -19721.539,E2 -19721.539} C_VEL
LIN {X 0,Y 235.071,Z 257.681,A -85,B 0,C 180,E1 -19725.612,E2 -19725.612} C_VEL
LIN {X 0,Y 234.97,Z 257.714,A -85,B 0,C 180,E1 -19729.211,E2 -19729.211} C_VEL
LIN {X 0,Y 234.897,Z 257.723,A -85,B 0,C 180,E1 -19732.892,E2 -19732.892} C_VEL
LIN {X 0,Y 234.896,Z 257.718,A -85,B 0,C 180,E1 -19736.669,E2 -19736.669} C_VEL
LIN {X 0,Y 234.871,Z 257.727,A -85,B 0,C 180,E1 -19740.579,E2 -19740.579} C_VEL
LIN {X 0,Y 234.898,Z 257.724,A -85,B 0,C 180,E1 -19744.646,E2 -19744.646} C_VEL
LIN {X 0,Y 234.891,Z 257.711,A -85,B 0,C 180,E1 -19748.942,E2 -19748.942} C_VEL
LIN {X 0,Y 234.833,Z 257.731,A -85,B 0,C 180,E1 -19753.502,E2 -19753.502} C_VEL
LIN {X 0,Y 234.835,Z 257.726,A -85,B 0,C 180,E1 -19756.513,E2 -19756.513} C_VEL
LIN {X 0,Y 234.904,Z 257.712,A -85,B 0,C 180,E1 -19761.086,E2 -19761.086} C_VEL
LIN {X 0,Y 234.912,Z 257.721,A -85,B 0,C 180,E1 -19765.369,E2 -19765.369} C_VEL
LIN {X 0,Y 234.885,Z 257.699,A -85,B 0,C 180,E1 -19769.435,E2 -19769.435} C_VEL
LIN {X 0,Y 234.933,Z 257.716,A -85,B 0,C 180,E1 -19773.83,E2 -19773.83} C_VEL
LIN {X 0,Y 234.936,Z 257.717,A -85,B 0,C 180,E1 -19778.971,E2 -19778.971} C_VEL
LIN {X 0,Y 235.055,Z 257.673,A -85,B 0,C 180,E1 -19783.101,E2 -19783.101} C_VEL
LIN {X 0,Y 235.111,Z 257.695,A -85,B 0,C 180,E1 -19787.929,E2 -19787.929} C_VEL
LIN {X 0,Y 235.315,Z 257.671,A -85,B 0,C 180,E1 -19791.419,E2 -19791.419} C_VEL
LIN {X 0,Y 235.352,Z 257.66,A -85,B 0,C 180,E1 -19793.147,E2 -19793.147} C_VEL
LIN {X 0,Y 235.583,Z 257.615,A -85,B 0,C 180,E1 -19798.297,E2 -19798.297} C_VEL
LIN {X 0,Y 235.584,Z 257.636,A -85,B 0,C 180,E1 -19801.716,E2 -19801.716} C_VEL
LIN {X 0,Y 235.352,Z 257.655,A -85,B 0,C 180,E1 -19806.867,E2 -19806.867} C_VEL
LIN {X 0,Y 235.199,Z 257.66,A -85,B 0,C 180,E1 -19810.335,E2 -19810.335} C_VEL
LIN {X 0,Y 235.089,Z 257.699,A -85,B 0,C 180,E1 -19815.614,E2 -19815.614} C_VEL
LIN {X 0,Y 234.971,Z 257.697,A -85,B 0,C 180,E1 -19819.422,E2 -19819.422} C_VEL
LIN {X 0,Y 234.954,Z 257.709,A -85,B 0,C 180,E1 -19822.89,E2 -19822.89} C_VEL
LIN {X 0,Y 234.946,Z 257.716,A -85,B 0,C 180,E1 -19826.863,E2 -19826.863} C_VEL
LIN {X 0,Y 234.214,Z 257.801,A -85,B 0,C 180,E1 -19828.293,E2 -19828.293} C_VEL
LIN {X 0,Y 231.364,Z 258.155,A -85,B 0,C 180,E1 -19830.629,E2 -19830.629} C_VEL
LIN {X 0,Y 228.976,Z 258.46,A -85,B 0,C 180,E1 -19832.532,E2 -19832.532} C_VEL
LIN {X 0,Y 227.944,Z 258.589,A -85,B 0,C 180,E1 -19834.009,E2 -19834.009} C_VEL
LIN {X 0,Y 227.853,Z 258.593,A -85,B 0,C 180,E1 -19834.509,E2 -19834.509} C_VEL
LIN {X 0,Y 227.857,Z 258.596,A -85,B 0,C 180,E1 -19838.095,E2 -19838.095} C_VEL
LIN {X 0,Y 227.804,Z 258.597,A -85,B 0,C 180,E1 -19842.751,E2 -19842.751} C_VEL
LIN {X 0,Y 227.83,Z 258.606,A -85,B 0,C 180,E1 -19845.201,E2 -19845.201} C_VEL
LIN {X 0,Y 227.821,Z 258.607,A -85,B 0,C 180,E1 -19849.619,E2 -19849.619} C_VEL
LIN {X 0,Y 227.915,Z 258.591,A -85,B 0,C 180,E1 -19854.403,E2 -19854.403} C_VEL
LIN {X 0,Y 227.996,Z 259.024,A -85,B 0,C 180,E1 -19854.957,E2 -19854.957} C_VEL
LIN {X 0,Y 229.663,Z 266.746,A -85,B 0,C 180,E1 -19858.279,E2 -19858.279} C_VEL
LIN {X 0,Y 231.23,Z 270.937,A -85,B 0,C 180,E1 -19858.713,E2 -19858.713} C_VEL
LIN {X 0,Y 238.172,Z 289.993,A -85,B 0,C 180,E1 -19860.124,E2 -19860.124} C_VEL
LIN {X 0,Y 241.577,Z 314.245,A -85,B 0,C 180,E1 -19861.267,E2 -19861.267} C_VEL
LIN {X 0,Y 239.47,Z 375.336,A -85,B 0,C 180,E1 -19863.116,E2 -19863.116} C_VEL
LIN {X 0,Y 238.473,Z 388.313,A -85,B 0,C 180,E1 -19863.821,E2 -19863.821} C_VEL
LIN {X 0,Y 237.213,Z 400.388,A -85,B 0,C 180,E1 -19864.79,E2 -19864.79} C_VEL
LIN {X 0,Y 235.693,Z 411.798,A -85,B 0,C 180,E1 -19866.026,E2 -19866.026} C_VEL
LIN {X 0,Y 234.08,Z 422.252,A -85,B 0,C 180,E1 -19867.49,E2 -19867.49} C_VEL
LIN {X 0,Y 232.368,Z 432.177,A -85,B 0,C 180,E1 -19869.227,E2 -19869.227} C_VEL
LIN {X 0,Y 230.748,Z 441.867,A -85,B 0,C 180,E1 -19871.346,E2 -19871.346} C_VEL
LIN {X 0,Y 229.213,Z 449.954,A -85,B 0,C 180,E1 -19873.521,E2 -19873.521} C_VEL
LIN {X 0,Y 227.693,Z 457.849,A -85,B 0,C 180,E1 -19876.157,E2 -19876.157} C_VEL
LIN {X 0,Y 226.862,Z 463.218,A -85,B 0,C 180,E1 -19878.381,E2 -19878.381} C_VEL
LIN {X 0,Y 226.151,Z 468.42,A -85,B 0,C 180,E1 -19881.058,E2 -19881.058} C_VEL
LIN {X 0,Y 225.721,Z 472.436,A -85,B 0,C 180,E1 -19883.741,E2 -19883.741} C_VEL
LIN {X 0,Y 225.569,Z 475.388,A -85,B 0,C 180,E1 -19886.425,E2 -19886.425} C_VEL
LIN {X 0,Y 225.581,Z 476.791,A -85,B 0,C 180,E1 -19888.212,E2 -19888.212} C_VEL
LIN {X 0,Y 225.646,Z 477.783,A -85,B 0,C 180,E1 -19889.997,E2 -19889.997} C_VEL
LIN {X 0,Y 225.579,Z 478.381,A -85,B 0,C 180,E1 -19891.783,E2 -19891.783} C_VEL
LIN {X 0,Y 225.655,Z 478.498,A -85,B 0,C 180,E1 -19894.643,E2 -19894.643} C_VEL
LIN {X 0,Y 225.942,Z 477.772,A -85,B 0,C 180,E1 -19897.144,E2 -19897.144} C_VEL
LIN {X 0,Y 226.869,Z 475.414,A -85,B 0,C 180,E1 -19900.709,E2 -19900.709} C_VEL
LIN {X 0,Y 228.046,Z 472.537,A -85,B 0,C 180,E1 -19903.361,E2 -19903.361} C_VEL
LIN {X 0,Y 229.626,Z 468.664,A -85,B 0,C 180,E1 -19905.986,E2 -19905.986} C_VEL
LIN {X 0,Y 231.828,Z 463.688,A -85,B 0,C 180,E1 -19908.558,E2 -19908.558} C_VEL
LIN {X 0,Y 234.423,Z 457.465,A -85,B 0,C 180,E1 -19911.082,E2 -19911.082} C_VEL
LIN {X 0,Y 237.292,Z 449.724,A -85,B 0,C 180,E1 -19913.565,E2 -19913.565} C_VEL
LIN {X 0,Y 240.189,Z 441.845,A -85,B 0,C 180,E1 -19915.565,E2 -19915.565} C_VEL
LIN {X 0,Y 243.639,Z 431.215,A -85,B 0,C 180,E1 -19917.716,E2 -19917.716} C_VEL
LIN {X 0,Y 246.736,Z 420.335,A -85,B 0,C 180,E1 -19919.426,E2 -19919.426} C_VEL
LIN {X 0,Y 249.785,Z 407.968,A -85,B 0,C 180,E1 -19920.893,E2 -19920.893} C_VEL
LIN {X 0,Y 252.156,Z 395.865,A -85,B 0,C 180,E1 -19921.973,E2 -19921.973} C_VEL
LIN {X 0,Y 254.025,Z 383.193,A -85,B 0,C 180,E1 -19922.764,E2 -19922.764} C_VEL
LIN {X 0,Y 255.263,Z 370.068,A -85,B 0,C 180,E1 -19923.29,E2 -19923.29} C_VEL
LIN {X 0,Y 257.654,Z 319.602,A -85,B 0,C 180,E1 -19924.736,E2 -19924.736} C_VEL
LIN {X 0,Y 256.641,Z 314.219,A -85,B 0,C 180,E1 -19925.138,E2 -19925.138} C_VEL
LIN {X 0,Y 250.884,Z 301.405,A -85,B 0,C 180,E1 -19926.835,E2 -19926.835} C_VEL
LIN {X 0,Y 244.413,Z 288.86,A -85,B 0,C 180,E1 -19928.842,E2 -19928.842} C_VEL
LIN {X 0,Y 239.359,Z 280.294,A -85,B 0,C 180,E1 -19930.485,E2 -19930.485} C_VEL
LIN {X 0,Y 235.599,Z 274.423,A -85,B 0,C 180,E1 -19931.768,E2 -19931.768} C_VEL
LIN {X 0,Y 233.066,Z 270.457,A -85,B 0,C 180,E1 -19932.692,E2 -19932.692} C_VEL
LIN {X 0,Y 230.048,Z 265.671,A -85,B 0,C 180,E1 -19933.953,E2 -19933.953} C_VEL
LIN {X 0,Y 228.204,Z 260.169,A -85,B 0,C 180,E1 -19937.652,E2 -19937.652} C_VEL
LIN {X 0,Y 227.813,Z 258.628,A -85,B 0,C 180,E1 -19938.979,E2 -19938.979} C_VEL
LIN {X 0,Y 227.88,Z 258.592,A -85,B 0,C 180,E1 -19943.303,E2 -19943.303} C_VEL
LIN {X 0,Y 227.88,Z 258.593,A -85,B 0,C 180,E1 -19946.371,E2 -19946.371} C_VEL
LIN {X 0,Y 227.876,Z 258.59,A -85,B 0,C 180,E1 -19950.425,E2 -19950.425} C_VEL
LIN {X 0,Y 227.87,Z 258.589,A -85,B 0,C 180,E1 -19954.412,E2 -19954.412} C_VEL
LIN {X 0,Y 227.917,Z 258.584,A -85,B 0,C 180,E1 -19958.276,E2 -19958.276} C_VEL
LIN {X 0,Y 228.012,Z 258.57,A -85,B 0,C 180,E1 -19963.888,E2 -19963.888} C_VEL
LIN {X 0,Y 228.048,Z 258.564,A -85,B 0,C 180,E1 -19967.535,E2 -19967.535} C_VEL
LIN {X 0,Y 228.245,Z 258.545,A -85,B 0,C 180,E1 -19971.137,E2 -19971.137} C_VEL
LIN {X 0,Y 228.292,Z 258.534,A -85,B 0,C 180,E1 -19972.92,E2 -19972.92} C_VEL
LIN {X 0,Y 228.521,Z 258.513,A -85,B 0,C 180,E1 -19978.231,E2 -19978.231} C_VEL
LIN {X 0,Y 228.521,Z 258.507,A -85,B 0,C 180,E1 -19981.755,E2 -19981.755} C_VEL
LIN {X 0,Y 228.283,Z 258.547,A -85,B 0,C 180,E1 -19987.066,E2 -19987.066} C_VEL
LIN {X 0,Y 228.124,Z 258.563,A -85,B 0,C 180,E1 -19990.645,E2 -19990.645} C_VEL
LIN {X 0,Y 228.019,Z 258.577,A -85,B 0,C 180,E1 -19994.267,E2 -19994.267} C_VEL
LIN {X 0,Y 227.933,Z 258.591,A -85,B 0,C 180,E1 -19997.951,E2 -19997.951} C_VEL
LIN {X 0,Y 227.916,Z 258.73,A -85,B 0,C 180,E1 -20002.584,E2 -20002.584} C_VEL
LIN {X 0,Y 228.966,Z 261.867,A -85,B 0,C 180,E1 -20004.774,E2 -20004.774} C_VEL
LIN {X 0,Y 232.462,Z 267.008,A -85,B 0,C 180,E1 -20006.193,E2 -20006.193} C_VEL
LIN {X 0,Y 237.004,Z 273.934,A -85,B 0,C 180,E1 -20007.834,E2 -20007.834} C_VEL
LIN {X 0,Y 242.317,Z 282.26,A -85,B 0,C 180,E1 -20009.596,E2 -20009.596} C_VEL
LIN {X 0,Y 248.829,Z 293.628,A -85,B 0,C 180,E1 -20011.626,E2 -20011.626} C_VEL
LIN {X 0,Y 255.09,Z 306.307,A -85,B 0,C 180,E1 -20013.487,E2 -20013.487} C_VEL
LIN {X 0,Y 258.073,Z 313.17,A -85,B 0,C 180,E1 -20014.34,E2 -20014.34} C_VEL
LIN {X 0,Y 255.031,Z 369.635,A -85,B 0,C 180,E1 -20015.94,E2 -20015.94} C_VEL
LIN {X 0,Y 253.469,Z 383.665,A -85,B 0,C 180,E1 -20016.649,E2 -20016.649} C_VEL
LIN {X 0,Y 251.495,Z 395.922,A -85,B 0,C 180,E1 -20017.578,E2 -20017.578} C_VEL
LIN {X 0,Y 249.051,Z 407.604,A -85,B 0,C 180,E1 -20018.785,E2 -20018.785} C_VEL
LIN {X 0,Y 246.301,Z 418.515,A -85,B 0,C 180,E1 -20020.25,E2 -20020.25} C_VEL
LIN {X 0,Y 243.329,Z 428.557,A -85,B 0,C 180,E1 -20021.954,E2 -20021.954} C_VEL
LIN {X 0,Y 240.552,Z 436.803,A -85,B 0,C 180,E1 -20023.694,E2 -20023.694} C_VEL
LIN {X 0,Y 237.415,Z 445.297,A -85,B 0,C 180,E1 -20025.925,E2 -20025.925} C_VEL
LIN {X 0,Y 234.203,Z 453.461,A -85,B 0,C 180,E1 -20028.69,E2 -20028.69} C_VEL
LIN {X 0,Y 231.532,Z 459.889,A -85,B 0,C 180,E1 -20031.523,E2 -20031.523} C_VEL
LIN {X 0,Y 229.376,Z 464.783,A -85,B 0,C 180,E1 -20034.402,E2 -20034.402} C_VEL
LIN {X 0,Y 227.78,Z 468.385,A -85,B 0,C 180,E1 -20037.323,E2 -20037.323} C_VEL
LIN {X 0,Y 226.573,Z 470.812,A -85,B 0,C 180,E1 -20040.269,E2 -20040.269} C_VEL
LIN {X 0,Y 225.975,Z 471.804,A -85,B 0,C 180,E1 -20042.195,E2 -20042.195} C_VEL
LIN {X 0,Y 225.465,Z 472.377,A -85,B 0,C 180,E1 -20044.663,E2 -20044.663} C_VEL
LIN {X 0,Y 225.144,Z 471.981,A -85,B 0,C 180,E1 -20048.004,E2 -20048.004} C_VEL
LIN {X 0,Y 225.176,Z 471.128,A -85,B 0,C 180,E1 -20049.924,E2 -20049.924} C_VEL
LIN {X 0,Y 225.213,Z 469.802,A -85,B 0,C 180,E1 -20051.82,E2 -20051.82} C_VEL
LIN {X 0,Y 225.644,Z 466.682,A -85,B 0,C 180,E1 -20054.88,E2 -20054.88} C_VEL
LIN {X 0,Y 226.172,Z 463.026,A -85,B 0,C 180,E1 -20057.44,E2 -20057.44} C_VEL
LIN {X 0,Y 226.966,Z 457.905,A -85,B 0,C 180,E1 -20060.197,E2 -20060.197} C_VEL
LIN {X 0,Y 228.028,Z 451.457,A -85,B 0,C 180,E1 -20062.921,E2 -20062.921} C_VEL
LIN {X 0,Y 229.489,Z 443.34,A -85,B 0,C 180,E1 -20065.612,E2 -20065.612} C_VEL
LIN {X 0,Y 231.008,Z 435.035,A -85,B 0,C 180,E1 -20067.823,E2 -20067.823} C_VEL
LIN {X 0,Y 232.936,Z 424.84,A -85,B 0,C 180,E1 -20070.003,E2 -20070.003} C_VEL
LIN {X 0,Y 234.65,Z 414.756,A -85,B 0,C 180,E1 -20071.719,E2 -20071.719} C_VEL
LIN {X 0,Y 236.207,Z 403.792,A -85,B 0,C 180,E1 -20073.201,E2 -20073.201} C_VEL
LIN {X 0,Y 237.676,Z 391.697,A -85,B 0,C 180,E1 -20074.454,E2 -20074.454} C_VEL
LIN {X 0,Y 238.885,Z 378.577,A -85,B 0,C 180,E1 -20075.436,E2 -20075.436} C_VEL
LIN {X 0,Y 239.661,Z 365.612,A -85,B 0,C 180,E1 -20076.052,E2 -20076.052} C_VEL
LIN {X 0,Y 241.758,Z 301.252,A -85,B 0,C 180,E1 -20077.98,E2 -20077.98} C_VEL
LIN {X 0,Y 240.319,Z 292.524,A -85,B 0,C 180,E1 -20078.411,E2 -20078.411} C_VEL
LIN {X 0,Y 232.661,Z 270.929,A -85,B 0,C 180,E1 -20079.962,E2 -20079.962} C_VEL
LIN {X 0,Y 228.784,Z 261.615,A -85,B 0,C 180,E1 -20080.77,E2 -20080.77} C_VEL
LIN {X 0,Y 228.542,Z 260.659,A -85,B 0,C 180,E1 -20081.04,E2 -20081.04} C_VEL
LIN {X 0,Y 228.047,Z 258.608,A -85,B 0,C 180,E1 -20082.088,E2 -20082.088} C_VEL
LIN {X 0,Y 228.02,Z 258.556,A -85,B 0,C 180,E1 -20086.108,E2 -20086.108} C_VEL
LIN {X 0,Y 227.901,Z 258.598,A -85,B 0,C 180,E1 -20089.832,E2 -20089.832} C_VEL
LIN {X 0,Y 227.842,Z 258.604,A -85,B 0,C 180,E1 -20093.643,E2 -20093.643} C_VEL
LIN {X 0,Y 227.816,Z 258.602,A -85,B 0,C 180,E1 -20097.567,E2 -20097.567} C_VEL
LIN {X 0,Y 227.83,Z 258.598,A -85,B 0,C 180,E1 -20101.631,E2 -20101.631} C_VEL
LIN {X 0,Y 227.842,Z 258.604,A -85,B 0,C 180,E1 -20105.882,E2 -20105.882} C_VEL
LIN {X 0,Y 227.779,Z 258.594,A -85,B 0,C 180,E1 -20110.39,E2 -20110.39} C_VEL
LIN {X 0,Y 227.792,Z 258.608,A -85,B 0,C 180,E1 -20115.207,E2 -20115.207} C_VEL
LIN {X 0,Y 227.785,Z 258.589,A -85,B 0,C 180,E1 -20119.625,E2 -20119.625} C_VEL
LIN {X 0,Y 227.852,Z 258.601,A -85,B 0,C 180,E1 -20124.133,E2 -20124.133} C_VEL
LIN {X 0,Y 227.844,Z 258.586,A -85,B 0,C 180,E1 -20128.383,E2 -20128.383} C_VEL
LIN {X 0,Y 227.825,Z 258.589,A -85,B 0,C 180,E1 -20132.446,E2 -20132.446} C_VEL
LIN {X 0,Y 227.86,Z 258.6,A -85,B 0,C 180,E1 -20136.37,E2 -20136.37} C_VEL
LIN {X 0,Y 227.893,Z 258.583,A -85,B 0,C 180,E1 -20140.178,E2 -20140.178} C_VEL
LIN {X 0,Y 228.018,Z 258.549,A -85,B 0,C 180,E1 -20143.903,E2 -20143.903} C_VEL
LIN {X 0,Y 228.066,Z 258.569,A -85,B 0,C 180,E1 -20147.55,E2 -20147.55} C_VEL
LIN {X 0,Y 228.257,Z 258.55,A -85,B 0,C 180,E1 -20151.151,E2 -20151.151} C_VEL
LIN {X 0,Y 228.305,Z 258.537,A -85,B 0,C 180,E1 -20152.934,E2 -20152.934} C_VEL
LIN {X 0,Y 228.541,Z 258.49,A -85,B 0,C 180,E1 -20158.245,E2 -20158.245} C_VEL
LIN {X 0,Y 228.542,Z 258.513,A -85,B 0,C 180,E1 -20161.769,E2 -20161.769} C_VEL
LIN {X 0,Y 228.304,Z 258.531,A -85,B 0,C 180,E1 -20167.08,E2 -20167.08} C_VEL
LIN {X 0,Y 228.141,Z 258.54,A -85,B 0,C 180,E1 -20170.658,E2 -20170.658} C_VEL
LIN {X 0,Y 228.048,Z 258.576,A -85,B 0,C 180,E1 -20174.28,E2 -20174.28} C_VEL
LIN {X 0,Y 227.946,Z 258.584,A -85,B 0,C 180,E1 -20177.964,E2 -20177.964} C_VEL
LIN {X 0,Y 227.92,Z 258.581,A -85,B 0,C 180,E1 -20182.317,E2 -20182.317} C_VEL
LIN {X 0,Y 227.919,Z 258.592,A -85,B 0,C 180,E1 -20186.825,E2 -20186.825} C_VEL
LIN {X 0,Y 227.875,Z 258.594,A -85,B 0,C 180,E1 -20191.628,E2 -20191.628} C_VEL
LIN {X 0,Y 227.853,Z 258.593,A -85,B 0,C 180,E1 -20194.509,E2 -20194.509} C_VEL
LIN {X 0,Y 227.162,Z 258.678,A -85,B 0,C 180,E1 -20195.985,E2 -20195.985} C_VEL
LIN {X 0,Y 224.296,Z 259.042,A -85,B 0,C 180,E1 -20198.394,E2 -20198.394} C_VEL
LIN {X 0,Y 221.873,Z 259.346,A -85,B 0,C 180,E1 -20200.36,E2 -20200.36} C_VEL
LIN {X 0,Y 220.838,Z 259.466,A -85,B 0,C 180,E1 -20201.886,E2 -20201.886} C_VEL
LIN {X 0,Y 220.755,Z 259.474,A -85,B 0,C 180,E1 -20202.403,E2 -20202.403} C_VEL
LIN {X 0,Y 220.764,Z 259.478,A -85,B 0,C 180,E1 -20207.079,E2 -20207.079} C_VEL
LIN {X 0,Y 220.802,Z 259.474,A -85,B 0,C 180,E1 -20210.459,E2 -20210.459} C_VEL
LIN {X 0,Y 220.879,Z 259.65,A -85,B 0,C 180,E1 -20214.218,E2 -20214.218} C_VEL
LIN {X 0,Y 222.425,Z 266.672,A -85,B 0,C 180,E1 -20217.404,E2 -20217.404} C_VEL
LIN {X 0,Y 224.527,Z 272.182,A -85,B 0,C 180,E1 -20217.958,E2 -20217.958} C_VEL
LIN {X 0,Y 231.336,Z 290.43,A -85,B 0,C 180,E1 -20219.398,E2 -20219.398} C_VEL
LIN {X 0,Y 232.351,Z 294.758,A -85,B 0,C 180,E1 -20219.659,E2 -20219.659} C_VEL
LIN {X 0,Y 234.983,Z 315.212,A -85,B 0,C 180,E1 -20220.634,E2 -20220.634} C_VEL
LIN {X 0,Y 232.888,Z 374.887,A -85,B 0,C 180,E1 -20222.475,E2 -20222.475} C_VEL
LIN {X 0,Y 231.859,Z 387.981,A -85,B 0,C 180,E1 -20223.197,E2 -20223.197} C_VEL
LIN {X 0,Y 230.488,Z 400.687,A -85,B 0,C 180,E1 -20224.243,E2 -20224.243} C_VEL
LIN {X 0,Y 228.924,Z 411.987,A -85,B 0,C 180,E1 -20225.512,E2 -20225.512} C_VEL
LIN {X 0,Y 227.446,Z 421.054,A -85,B 0,C 180,E1 -20226.795,E2 -20226.795} C_VEL
LIN {X 0,Y 225.699,Z 431.195,A -85,B 0,C 180,E1 -20228.583,E2 -20228.583} C_VEL
LIN {X 0,Y 223.895,Z 441.366,A -85,B 0,C 180,E1 -20230.842,E2 -20230.842} C_VEL
LIN {X 0,Y 222.092,Z 450.736,A -85,B 0,C 180,E1 -20233.45,E2 -20233.45} C_VEL
LIN {X 0,Y 220.555,Z 458.421,A -85,B 0,C 180,E1 -20236.17,E2 -20236.17} C_VEL
LIN {X 0,Y 219.591,Z 464.598,A -85,B 0,C 180,E1 -20238.926,E2 -20238.926} C_VEL
LIN {X 0,Y 218.916,Z 469.471,A -85,B 0,C 180,E1 -20241.691,E2 -20241.691} C_VEL
LIN {X 0,Y 218.586,Z 473.196,A -85,B 0,C 180,E1 -20244.462,E2 -20244.462} C_VEL
LIN {X 0,Y 218.471,Z 475.11,A -85,B 0,C 180,E1 -20246.308,E2 -20246.308} C_VEL
LIN {X 0,Y 218.484,Z 476.577,A -85,B 0,C 180,E1 -20248.154,E2 -20248.154} C_VEL
LIN {X 0,Y 218.564,Z 477.603,A -85,B 0,C 180,E1 -20249.997,E2 -20249.997} C_VEL
LIN {X 0,Y 218.482,Z 478.232,A -85,B 0,C 180,E1 -20251.84,E2 -20251.84} C_VEL
LIN {X 0,Y 218.649,Z 478.328,A -85,B 0,C 180,E1 -20255.531,E2 -20255.531} C_VEL
LIN {X 0,Y 219.311,Z 476.811,A -85,B 0,C 180,E1 -20259.217,E2 -20259.217} C_VEL
LIN {X 0,Y 220.651,Z 473.739,A -85,B 0,C 180,E1 -20262.88,E2 -20262.88} C_VEL
LIN {X 0,Y 222.196,Z 470.289,A -85,B 0,C 180,E1 -20265.593,E2 -20265.593} C_VEL
LIN {X 0,Y 224.295,Z 465.778,A -85,B 0,C 180,E1 -20268.257,E2 -20268.257} C_VEL
LIN {X 0,Y 227.4,Z 458.971,A -85,B 0,C 180,E1 -20271.29,E2 -20271.29} C_VEL
LIN {X 0,Y 230.29,Z 451.637,A -85,B 0,C 180,E1 -20273.848,E2 -20273.848} C_VEL
LIN {X 0,Y 233.146,Z 444.182,A -85,B 0,C 180,E1 -20275.915,E2 -20275.915} C_VEL
LIN {X 0,Y 236.794,Z 434.169,A -85,B 0,C 180,E1 -20278.107,E2 -20278.107} C_VEL
LIN {X 0,Y 239.921,Z 423.985,A -85,B 0,C 180,E1 -20279.863,E2 -20279.863} C_VEL
LIN {X 0,Y 243.014,Z 412.712,A -85,B 0,C 180,E1 -20281.367,E2 -20281.367} C_VEL
LIN {X 0,Y 245.624,Z 401.038,A -85,B 0,C 180,E1 -20282.563,E2 -20282.563} C_VEL
LIN {X 0,Y 247.809,Z 388.258,A -85,B 0,C 180,E1 -20283.511,E2 -20283.511} C_VEL
LIN {X 0,Y 249.48,Z 374.734,A -85,B 0,C 180,E1 -20284.167,E2 -20284.167} C_VEL
LIN {X 0,Y 252.284,Z 320.701,A -85,B 0,C 180,E1 -20285.765,E2 -20285.765} C_VEL
LIN {X 0,Y 251.635,Z 317.505,A -85,B 0,C 180,E1 -20286.028,E2 -20286.028} C_VEL
LIN {X 0,Y 246.506,Z 305.801,A -85,B 0,C 180,E1 -20287.633,E2 -20287.633} C_VEL
LIN {X 0,Y 240.426,Z 293.776,A -85,B 0,C 180,E1 -20289.609,E2 -20289.609} C_VEL
LIN {X 0,Y 235.49,Z 285.259,A -85,B 0,C 180,E1 -20291.288,E2 -20291.288} C_VEL
LIN {X 0,Y 232.344,Z 280.213,A -85,B 0,C 180,E1 -20292.428,E2 -20292.428} C_VEL
LIN {X 0,Y 229.4,Z 275.588,A -85,B 0,C 180,E1 -20293.545,E2 -20293.545} C_VEL
LIN {X 0,Y 226.015,Z 270.575,A -85,B 0,C 180,E1 -20294.89,E2 -20294.89} C_VEL
LIN {X 0,Y 222.694,Z 265.542,A -85,B 0,C 180,E1 -20296.395,E2 -20296.395} C_VEL
LIN {X 0,Y 220.823,Z 259.744,A -85,B 0,C 180,E1 -20300.755,E2 -20300.755} C_VEL
LIN {X 0,Y 220.828,Z 259.474,A -85,B 0,C 180,E1 -20302.787,E2 -20302.787} C_VEL
LIN {X 0,Y 220.813,Z 259.47,A -85,B 0,C 180,E1 -20307.236,E2 -20307.236} C_VEL
LIN {X 0,Y 220.799,Z 259.472,A -85,B 0,C 180,E1 -20311.474,E2 -20311.474} C_VEL
LIN {X 0,Y 220.801,Z 259.472,A -85,B 0,C 180,E1 -20315.551,E2 -20315.551} C_VEL
LIN {X 0,Y 220.847,Z 259.463,A -85,B 0,C 180,E1 -20319.503,E2 -20319.503} C_VEL
LIN {X 0,Y 220.971,Z 259.446,A -85,B 0,C 180,E1 -20323.36,E2 -20323.36} C_VEL
LIN {X 0,Y 221.054,Z 259.44,A -85,B 0,C 180,E1 -20328.996,E2 -20328.996} C_VEL
LIN {X 0,Y 221.23,Z 259.412,A -85,B 0,C 180,E1 -20332.693,E2 -20332.693} C_VEL
LIN {X 0,Y 221.454,Z 259.392,A -85,B 0,C 180,E1 -20338.174,E2 -20338.174} C_VEL
LIN {X 0,Y 221.454,Z 259.387,A -85,B 0,C 180,E1 -20341.812,E2 -20341.812} C_VEL
LIN {X 0,Y 221.221,Z 259.428,A -85,B 0,C 180,E1 -20347.293,E2 -20347.293} C_VEL
LIN {X 0,Y 221.045,Z 259.448,A -85,B 0,C 180,E1 -20350.99,E2 -20350.99} C_VEL
LIN {X 0,Y 220.959,Z 259.453,A -85,B 0,C 180,E1 -20356.626,E2 -20356.626} C_VEL
LIN {X 0,Y 220.879,Z 259.645,A -85,B 0,C 180,E1 -20360.479,E2 -20360.479} C_VEL
LIN {X 0,Y 221.769,Z 262.155,A -85,B 0,C 180,E1 -20362.343,E2 -20362.343} C_VEL
LIN {X 0,Y 224.449,Z 266.231,A -85,B 0,C 180,E1 -20363.587,E2 -20363.587} C_VEL
LIN {X 0,Y 226.214,Z 268.454,A -85,B 0,C 180,E1 -20364.3,E2 -20364.3} C_VEL
LIN {X 0,Y 230.564,Z 274.773,A -85,B 0,C 180,E1 -20366.007,E2 -20366.007} C_VEL
LIN {X 0,Y 235.993,Z 283.25,A -85,B 0,C 180,E1 -20367.994,E2 -20367.994} C_VEL
LIN {X 0,Y 242.87,Z 294.977,A -85,B 0,C 180,E1 -20370.285,E2 -20370.285} C_VEL
LIN {X 0,Y 249.115,Z 307.393,A -85,B 0,C 180,E1 -20372.255,E2 -20372.255} C_VEL
LIN {X 0,Y 252.611,Z 315.343,A -85,B 0,C 180,E1 -20373.328,E2 -20373.328} C_VEL
LIN {X 0,Y 249.615,Z 369.633,A -85,B 0,C 180,E1 -20374.904,E2 -20374.904} C_VEL
LIN {X 0,Y 248.115,Z 382.816,A -85,B 0,C 180,E1 -20375.568,E2 -20375.568} C_VEL
LIN {X 0,Y 245.986,Z 395.7,A -85,B 0,C 180,E1 -20376.534,E2 -20376.534} C_VEL
LIN {X 0,Y 243.273,Z 408.1,A -85,B 0,C 180,E1 -20377.834,E2 -20377.834} C_VEL
LIN {X 0,Y 240.124,Z 419.951,A -85,B 0,C 180,E1 -20379.476,E2 -20379.476} C_VEL
LIN {X 0,Y 236.626,Z 430.891,A -85,B 0,C 180,E1 -20381.454,E2 -20381.454} C_VEL
LIN {X 0,Y 233.152,Z 440.455,A -85,B 0,C 180,E1 -20383.665,E2 -20383.665} C_VEL
LIN {X 0,Y 230.02,Z 448.315,A -85,B 0,C 180,E1 -20385.969,E2 -20385.969} C_VEL
LIN {X 0,Y 227.136,Z 455.09,A -85,B 0,C 180,E1 -20388.495,E2 -20388.495} C_VEL
LIN {X 0,Y 224.294,Z 461.393,A -85,B 0,C 180,E1 -20391.554,E2 -20391.554} C_VEL
LIN {X 0,Y 222.335,Z 465.539,A -85,B 0,C 180,E1 -20394.216,E2 -20394.216} C_VEL
LIN {X 0,Y 220.687,Z 468.954,A -85,B 0,C 180,E1 -20397.226,E2 -20397.226} C_VEL
LIN {X 0,Y 219.621,Z 470.899,A -85,B 0,C 180,E1 -20399.752,E2 -20399.752} C_VEL
LIN {X 0,Y 218.631,Z 472.336,A -85,B 0,C 180,E1 -20403.257,E2 -20403.257} C_VEL
LIN {X 0,Y 218.271,Z 472.523,A -85,B 0,C 180,E1 -20405.258,E2 -20405.258} C_VEL
LIN {X 0,Y 218.069,Z 472.221,A -85,B 0,C 180,E1 -20407.252,E2 -20407.252} C_VEL
LIN {X 0,Y 218.064,Z 471.49,A -85,B 0,C 180,E1 -20409.239,E2 -20409.239} C_VEL
LIN {X 0,Y 218.091,Z 470.309,A -85,B 0,C 180,E1 -20411.204,E2 -20411.204} C_VEL
LIN {X 0,Y 218.507,Z 466.943,A -85,B 0,C 180,E1 -20414.742,E2 -20414.742} C_VEL
LIN {X 0,Y 219.205,Z 462.42,A -85,B 0,C 180,E1 -20417.975,E2 -20417.975} C_VEL
LIN {X 0,Y 220.072,Z 457.101,A -85,B 0,C 180,E1 -20420.815,E2 -20420.815} C_VEL
LIN {X 0,Y 221.217,Z 450.376,A -85,B 0,C 180,E1 -20423.619,E2 -20423.619} C_VEL
LIN {X 0,Y 222.867,Z 441.972,A -85,B 0,C 180,E1 -20426.387,E2 -20426.387} C_VEL
LIN {X 0,Y 224.386,Z 433.841,A -85,B 0,C 180,E1 -20428.544,E2 -20428.544} C_VEL
LIN {X 0,Y 226.278,Z 423.901,A -85,B 0,C 180,E1 -20430.67,E2 -20430.67} C_VEL
LIN {X 0,Y 228.276,Z 412.088,A -85,B 0,C 180,E1 -20432.65,E2 -20432.65} C_VEL
LIN {X 0,Y 229.92,Z 400.464,A -85,B 0,C 180,E1 -20434.166,E2 -20434.166} C_VEL
LIN {X 0,Y 231.341,Z 388.383,A -85,B 0,C 180,E1 -20435.341,E2 -20435.341} C_VEL
LIN {X 0,Y 232.503,Z 375.317,A -85,B 0,C 180,E1 -20436.239,E2 -20436.239} C_VEL
LIN {X 0,Y 233.273,Z 361.542,A -85,B 0,C 180,E1 -20436.816,E2 -20436.816} C_VEL
LIN {X 0,Y 235.292,Z 302.703,A -85,B 0,C 180,E1 -20438.592,E2 -20438.592} C_VEL
LIN {X 0,Y 233.984,Z 294.73,A -85,B 0,C 180,E1 -20439.001,E2 -20439.001} C_VEL
LIN {X 0,Y 226.653,Z 273.856,A -85,B 0,C 180,E1 -20440.558,E2 -20440.558} C_VEL
LIN {X 0,Y 221.54,Z 261.748,A -85,B 0,C 180,E1 -20441.667,E2 -20441.667} C_VEL
LIN {X 0,Y 221.057,Z 259.742,A -85,B 0,C 180,E1 -20442.441,E2 -20442.441} C_VEL
LIN {X 0,Y 220.976,Z 259.455,A -85,B 0,C 180,E1 -20442.866,E2 -20442.866} C_VEL
LIN {X 0,Y 220.952,Z 259.438,A -85,B 0,C 180,E1 -20447.432,E2 -20447.432} C_VEL
LIN {X 0,Y 220.825,Z 259.473,A -85,B 0,C 180,E1 -20452.455,E2 -20452.455} C_VEL
LIN {X 0,Y 220.822,Z 259.471,A -85,B 0,C 180,E1 -20457.003,E2 -20457.003} C_VEL
LIN {X 0,Y 220.794,Z 259.479,A -85,B 0,C 180,E1 -20460.765,E2 -20460.765} C_VEL
LIN {X 0,Y 220.77,Z 259.485,A -85,B 0,C 180,E1 -20464.964,E2 -20464.964} C_VEL
LIN {X 0,Y 220.78,Z 259.48,A -85,B 0,C 180,E1 -20467.282,E2 -20467.282} C_VEL
LIN {X 0,Y 220.728,Z 259.482,A -85,B 0,C 180,E1 -20471.966,E2 -20471.966} C_VEL
LIN {X 0,Y 220.735,Z 259.486,A -85,B 0,C 180,E1 -20475.548,E2 -20475.548} C_VEL
LIN {X 0,Y 220.767,Z 259.466,A -85,B 0,C 180,E1 -20480.466,E2 -20480.466} C_VEL
LIN {X 0,Y 220.813,Z 259.476,A -85,B 0,C 180,E1 -20482.801,E2 -20482.801} C_VEL
LIN {X 0,Y 220.801,Z 259.469,A -85,B 0,C 180,E1 -20487.251,E2 -20487.251} C_VEL
LIN {X 0,Y 220.784,Z 259.455,A -85,B 0,C 180,E1 -20491.488,E2 -20491.488} C_VEL
LIN {X 0,Y 220.797,Z 259.482,A -85,B 0,C 180,E1 -20495.566,E2 -20495.566} C_VEL
LIN {X 0,Y 220.848,Z 259.464,A -85,B 0,C 180,E1 -20499.518,E2 -20499.518} C_VEL
LIN {X 0,Y 220.976,Z 259.422,A -85,B 0,C 180,E1 -20503.375,E2 -20503.375} C_VEL
LIN {X 0,Y 221.002,Z 259.446,A -85,B 0,C 180,E1 -20507.146,E2 -20507.146} C_VEL
LIN {X 0,Y 221.198,Z 259.429,A -85,B 0,C 180,E1 -20510.867,E2 -20510.867} C_VEL
LIN {X 0,Y 221.243,Z 259.417,A -85,B 0,C 180,E1 -20512.707,E2 -20512.707} C_VEL
LIN {X 0,Y 221.474,Z 259.368,A -85,B 0,C 180,E1 -20518.189,E2 -20518.189} C_VEL
LIN {X 0,Y 221.475,Z 259.393,A -85,B 0,C 180,E1 -20521.825,E2 -20521.825} C_VEL
LIN {X 0,Y 221.242,Z 259.41,A -85,B 0,C 180,E1 -20527.307,E2 -20527.307} C_VEL
LIN {X 0,Y 221.067,Z 259.424,A -85,B 0,C 180,E1 -20531.003,E2 -20531.003} C_VEL
LIN {X 0,Y 220.979,Z 259.46,A -85,B 0,C 180,E1 -20534.747,E2 -20534.747} C_VEL
LIN {X 0,Y 220.886,Z 259.456,A -85,B 0,C 180,E1 -20538.559,E2 -20538.559} C_VEL
LIN {X 0,Y 220.861,Z 259.461,A -85,B 0,C 180,E1 -20542.654,E2 -20542.654} C_VEL
LIN {X 0,Y 220.883,Z 259.466,A -85,B 0,C 180,E1 -20547.009,E2 -20547.009} C_VEL
LIN {X 0,Y 220.838,Z 259.462,A -85,B 0,C 180,E1 -20550.762,E2 -20550.762} C_VEL
LIN {X 0,Y 220.811,Z 259.475,A -85,B 0,C 180,E1 -20554.96,E2 -20554.96} C_VEL
LIN {X 0,Y 220.816,Z 259.466,A -85,B 0,C 180,E1 -20557.276,E2 -20557.276} C_VEL
LIN {X 0,Y 220.764,Z 259.475,A -85,B 0,C 180,E1 -20561.961,E2 -20561.961} C_VEL
LIN {X 0,Y 220.755,Z 259.474,A -85,B 0,C 180,E1 -20562.403,E2 -20562.403} C_VEL
LIN {X 0,Y 220.083,Z 259.567,A -85,B 0,C 180,E1 -20563.924,E2 -20563.924} C_VEL
LIN {X 0,Y 217.21,Z 259.923,A -85,B 0,C 180,E1 -20566.406,E2 -20566.406} C_VEL
LIN {X 0,Y 214.782,Z 260.228,A -85,B 0,C 180,E1 -20568.432,E2 -20568.432} C_VEL
LIN {X 0,Y 213.76,Z 260.354,A -85,B 0,C 180,E1 -20570.007,E2 -20570.007} C_VEL
LIN {X 0,Y 213.688,Z 260.353,A -85,B 0,C 180,E1 -20570.541,E2 -20570.541} C_VEL
LIN {X 0,Y 213.813,Z 260.493,A -85,B 0,C 180,E1 -20573.581,E2 -20573.581} C_VEL
LIN {X 0,Y 215.191,Z 266.543,A -85,B 0,C 180,E1 -20576.457,E2 -20576.457} C_VEL
LIN {X 0,Y 217.745,Z 273.041,A -85,B 0,C 180,E1 -20577.126,E2 -20577.126} C_VEL
LIN {X 0,Y 224.051,Z 289.72,A -85,B 0,C 180,E1 -20578.529,E2 -20578.529} C_VEL
LIN {X 0,Y 225.869,Z 295.551,A -85,B 0,C 180,E1 -20578.952,E2 -20578.952} C_VEL
LIN {X 0,Y 228.447,Z 315.5,A -85,B 0,C 180,E1 -20579.944,E2 -20579.944} C_VEL
LIN {X 0,Y 226.277,Z 374.944,A -85,B 0,C 180,E1 -20581.837,E2 -20581.837} C_VEL
LIN {X 0,Y 225.207,Z 388.171,A -85,B 0,C 180,E1 -20582.591,E2 -20582.591} C_VEL
LIN {X 0,Y 223.786,Z 400.798,A -85,B 0,C 180,E1 -20583.664,E2 -20583.664} C_VEL
LIN {X 0,Y 222.173,Z 412.039,A -85,B 0,C 180,E1 -20584.967,E2 -20584.967} C_VEL
LIN {X 0,Y 220.649,Z 421.086,A -85,B 0,C 180,E1 -20586.286,E2 -20586.286} C_VEL
LIN {X 0,Y 218.885,Z 430.984,A -85,B 0,C 180,E1 -20588.08,E2 -20588.08} C_VEL
LIN {X 0,Y 217.055,Z 440.814,A -85,B 0,C 180,E1 -20590.312,E2 -20590.312} C_VEL
LIN {X 0,Y 215.214,Z 449.973,A -85,B 0,C 180,E1 -20592.905,E2 -20592.905} C_VEL
LIN {X 0,Y 213.632,Z 457.82,A -85,B 0,C 180,E1 -20595.713,E2 -20595.713} C_VEL
LIN {X 0,Y 212.576,Z 464.092,A -85,B 0,C 180,E1 -20598.556,E2 -20598.556} C_VEL
LIN {X 0,Y 211.876,Z 469.054,A -85,B 0,C 180,E1 -20601.413,E2 -20601.413} C_VEL
LIN {X 0,Y 211.51,Z 472.859,A -85,B 0,C 180,E1 -20604.276,E2 -20604.276} C_VEL
LIN {X 0,Y 211.396,Z 474.812,A -85,B 0,C 180,E1 -20606.185,E2 -20606.185} C_VEL
LIN {X 0,Y 211.389,Z 476.341,A -85,B 0,C 180,E1 -20608.092,E2 -20608.092} C_VEL
LIN {X 0,Y 211.464,Z 477.413,A -85,B 0,C 180,E1 -20609.997,E2 -20609.997} C_VEL
LIN {X 0,Y 211.387,Z 478.079,A -85,B 0,C 180,E1 -20611.902,E2 -20611.902} C_VEL
LIN {X 0,Y 211.437,Z 478.39,A -85,B 0,C 180,E1 -20614.238,E2 -20614.238} C_VEL
LIN {X 0,Y 211.842,Z 477.751,A -85,B 0,C 180,E1 -20617.623,E2 -20617.623} C_VEL
LIN {X 0,Y 212.896,Z 475.543,A -85,B 0,C 180,E1 -20621.421,E2 -20621.421} C_VEL
LIN {X 0,Y 214.245,Z 472.819,A -85,B 0,C 180,E1 -20624.239,E2 -20624.239} C_VEL
LIN {X 0,Y 216.013,Z 469.106,A -85,B 0,C 180,E1 -20627.023,E2 -20627.023} C_VEL
LIN {X 0,Y 218.445,Z 464.299,A -85,B 0,C 180,E1 -20629.741,E2 -20629.741} C_VEL
LIN {X 0,Y 221.26,Z 458.266,A -85,B 0,C 180,E1 -20632.402,E2 -20632.402} C_VEL
LIN {X 0,Y 224.409,Z 450.799,A -85,B 0,C 180,E1 -20635.008,E2 -20635.008} C_VEL
LIN {X 0,Y 227.537,Z 443.187,A -85,B 0,C 180,E1 -20637.099,E2 -20637.099} C_VEL
LIN {X 0,Y 230.936,Z 433.964,A -85,B 0,C 180,E1 -20639.135,E2 -20639.135} C_VEL
LIN {X 0,Y 234.585,Z 422.5,A -85,B 0,C 180,E1 -20641.114,E2 -20641.114} C_VEL
LIN {X 0,Y 237.868,Z 410.918,A -85,B 0,C 180,E1 -20642.626,E2 -20642.626} C_VEL
LIN {X 0,Y 240.618,Z 398.617,A -85,B 0,C 180,E1 -20643.83,E2 -20643.83} C_VEL
LIN {X 0,Y 242.831,Z 385.759,A -85,B 0,C 180,E1 -20644.732,E2 -20644.732} C_VEL
LIN {X 0,Y 244.278,Z 373.257,A -85,B 0,C 180,E1 -20645.316,E2 -20645.316} C_VEL
LIN {X 0,Y 247.094,Z 322.322,A -85,B 0,C 180,E1 -20646.817,E2 -20646.817} C_VEL
LIN {X 0,Y 246.334,Z 319.7,A -85,B 0,C 180,E1 -20647.095,E2 -20647.095} C_VEL
LIN {X 0,Y 240.805,Z 307.231,A -85,B 0,C 180,E1 -20648.922,E2 -20648.922} C_VEL
LIN {X 0,Y 234.583,Z 295.173,A -85,B 0,C 180,E1 -20651.071,E2 -20651.071} C_VEL
LIN {X 0,Y 229.167,Z 285.968,A -85,B 0,C 180,E1 -20653.093,E2 -20653.093} C_VEL
LIN {X 0,Y 225.701,Z 280.567,A -85,B 0,C 180,E1 -20654.462,E2 -20654.462} C_VEL
LIN {X 0,Y 222.789,Z 276.143,A -85,B 0,C 180,E1 -20655.676,E2 -20655.676} C_VEL
LIN {X 0,Y 218.808,Z 270.481,A -85,B 0,C 180,E1 -20657.428,E2 -20657.428} C_VEL
LIN {X 0,Y 215.429,Z 265.705,A -85,B 0,C 180,E1 -20659.103,E2 -20659.103} C_VEL
LIN {X 0,Y 214.792,Z 263.846,A -85,B 0,C 180,E1 -20660.347,E2 -20660.347} C_VEL
LIN {X 0,Y 213.735,Z 260.382,A -85,B 0,C 180,E1 -20663.589,E2 -20663.589} C_VEL
LIN {X 0,Y 213.76,Z 260.353,A -85,B 0,C 180,E1 -20668.254,E2 -20668.254} C_VEL
LIN {X 0,Y 213.783,Z 260.356,A -85,B 0,C 180,E1 -20672.59,E2 -20672.59} C_VEL
LIN {X 0,Y 213.792,Z 260.355,A -85,B 0,C 180,E1 -20676.982,E2 -20676.982} C_VEL
LIN {X 0,Y 213.88,Z 260.33,A -85,B 0,C 180,E1 -20682.791,E2 -20682.791} C_VEL
LIN {X 0,Y 213.926,Z 260.327,A -85,B 0,C 180,E1 -20686.698,E2 -20686.698} C_VEL
LIN {X 0,Y 214.126,Z 260.31,A -85,B 0,C 180,E1 -20690.548,E2 -20690.548} C_VEL
LIN {X 0,Y 214.062,Z 260.32,A -85,B 0,C 180,E1 -20694.34,E2 -20694.34} C_VEL
LIN {X 0,Y 214.391,Z 260.27,A -85,B 0,C 180,E1 -20698.114,E2 -20698.114} C_VEL
LIN {X 0,Y 214.497,Z 260.26,A -85,B 0,C 180,E1 -20699.993,E2 -20699.993} C_VEL
LIN {X 0,Y 214.391,Z 260.267,A -85,B 0,C 180,E1 -20701.871,E2 -20701.871} C_VEL
LIN {X 0,Y 214.163,Z 260.309,A -85,B 0,C 180,E1 -20707.535,E2 -20707.535} C_VEL
LIN {X 0,Y 213.976,Z 260.332,A -85,B 0,C 180,E1 -20711.358,E2 -20711.358} C_VEL
LIN {X 0,Y 213.884,Z 260.343,A -85,B 0,C 180,E1 -20715.232,E2 -20715.232} C_VEL
LIN {X 0,Y 213.859,Z 260.47,A -85,B 0,C 180,E1 -20717.969,E2 -20717.969} C_VEL
LIN {X 0,Y 214.406,Z 262.441,A -85,B 0,C 180,E1 -20719.499,E2 -20719.499} C_VEL
LIN {X 0,Y 218.133,Z 267.386,A -85,B 0,C 180,E1 -20721.367,E2 -20721.367} C_VEL
LIN {X 0,Y 219.765,Z 269.769,A -85,B 0,C 180,E1 -20722.125,E2 -20722.125} C_VEL
LIN {X 0,Y 223.302,Z 274.489,A -85,B 0,C 180,E1 -20723.647,E2 -20723.647} C_VEL
LIN {X 0,Y 227.332,Z 280.465,A -85,B 0,C 180,E1 -20725.293,E2 -20725.293} C_VEL
LIN {X 0,Y 232.244,Z 288.239,A -85,B 0,C 180,E1 -20727.169,E2 -20727.169} C_VEL
LIN {X 0,Y 238.781,Z 299.705,A -85,B 0,C 180,E1 -20729.477,E2 -20729.477} C_VEL
LIN {X 0,Y 244.672,Z 311.651,A -85,B 0,C 180,E1 -20731.426,E2 -20731.426} C_VEL
LIN {X 0,Y 247.354,Z 317.894,A -85,B 0,C 180,E1 -20732.295,E2 -20732.295} C_VEL
LIN {X 0,Y 244.272,Z 370.091,A -85,B 0,C 180,E1 -20733.828,E2 -20733.828} C_VEL
LIN {X 0,Y 242.606,Z 383.806,A -85,B 0,C 180,E1 -20734.538,E2 -20734.538} C_VEL
LIN {X 0,Y 240.496,Z 395.907,A -85,B 0,C 180,E1 -20735.473,E2 -20735.473} C_VEL
LIN {X 0,Y 237.676,Z 408.224,A -85,B 0,C 180,E1 -20736.784,E2 -20736.784} C_VEL
LIN {X 0,Y 234.411,Z 420.007,A -85,B 0,C 180,E1 -20738.444,E2 -20738.444} C_VEL
LIN {X 0,Y 230.79,Z 430.816,A -85,B 0,C 180,E1 -20740.426,E2 -20740.426} C_VEL
LIN {X 0,Y 227.096,Z 440.545,A -85,B 0,C 180,E1 -20742.712,E2 -20742.712} C_VEL
LIN {X 0,Y 223.809,Z 448.371,A -85,B 0,C 180,E1 -20745.05,E2 -20745.05} C_VEL
LIN {X 0,Y 220.393,Z 455.899,A -85,B 0,C 180,E1 -20747.964,E2 -20747.964} C_VEL
LIN {X 0,Y 217.754,Z 461.437,A -85,B 0,C 180,E1 -20750.755,E2 -20750.755} C_VEL
LIN {X 0,Y 215.295,Z 466.294,A -85,B 0,C 180,E1 -20754.018,E2 -20754.018} C_VEL
LIN {X 0,Y 214.12,Z 468.554,A -85,B 0,C 180,E1 -20756.087,E2 -20756.087} C_VEL
LIN {X 0,Y 212.708,Z 470.98,A -85,B 0,C 180,E1 -20759.193,E2 -20759.193} C_VEL
LIN {X 0,Y 211.745,Z 472.308,A -85,B 0,C 180,E1 -20762.315,E2 -20762.315} C_VEL
LIN {X 0,Y 211.324,Z 472.612,A -85,B 0,C 180,E1 -20764.387,E2 -20764.387} C_VEL
LIN {X 0,Y 211.038,Z 472.457,A -85,B 0,C 180,E1 -20766.449,E2 -20766.449} C_VEL
LIN {X 0,Y 210.929,Z 471.658,A -85,B 0,C 180,E1 -20768.871,E2 -20768.871} C_VEL
LIN {X 0,Y 210.967,Z 470.746,A -85,B 0,C 180,E1 -20770.544,E2 -20770.544} C_VEL
LIN {X 0,Y 211.204,Z 468.274,A -85,B 0,C 180,E1 -20773.573,E2 -20773.573} C_VEL
LIN {X 0,Y 211.784,Z 464.724,A -85,B 0,C 180,E1 -20776.571,E2 -20776.571} C_VEL
LIN {X 0,Y 212.541,Z 460.031,A -85,B 0,C 180,E1 -20779.525,E2 -20779.525} C_VEL
LIN {X 0,Y 213.547,Z 454.042,A -85,B 0,C 180,E1 -20782.438,E2 -20782.438} C_VEL
LIN {X 0,Y 214.93,Z 446.532,A -85,B 0,C 180,E1 -20785.314,E2 -20785.314} C_VEL
LIN {X 0,Y 216.566,Z 438.832,A -85,B 0,C 180,E1 -20787.678,E2 -20787.678} C_VEL
LIN {X 0,Y 218.36,Z 429.52,A -85,B 0,C 180,E1 -20790.003,E2 -20790.003} C_VEL
LIN {X 0,Y 220.326,Z 419.129,A -85,B 0,C 180,E1 -20792.059,E2 -20792.059} C_VEL
LIN {X 0,Y 222.223,Z 407.566,A -85,B 0,C 180,E1 -20793.856,E2 -20793.856} C_VEL
LIN {X 0,Y 223.858,Z 395.577,A -85,B 0,C 180,E1 -20795.294,E2 -20795.294} C_VEL
LIN {X 0,Y 225.274,Z 383.007,A -85,B 0,C 180,E1 -20796.384,E2 -20796.384} C_VEL
LIN {X 0,Y 226.294,Z 369.27,A -85,B 0,C 180,E1 -20797.187,E2 -20797.187} C_VEL
LIN {X 0,Y 228.754,Z 303.349,A -85,B 0,C 180,E1 -20799.278,E2 -20799.278} C_VEL
LIN {X 0,Y 227.649,Z 296.788,A -85,B 0,C 180,E1 -20799.632,E2 -20799.632} C_VEL
LIN {X 0,Y 220.638,Z 276.699,A -85,B 0,C 180,E1 -20801.195,E2 -20801.195} C_VEL
LIN {X 0,Y 214.321,Z 261.925,A -85,B 0,C 180,E1 -20802.625,E2 -20802.625} C_VEL
LIN {X 0,Y 213.948,Z 260.506,A -85,B 0,C 180,E1 -20803.134,E2 -20803.134} C_VEL
LIN {X 0,Y 213.901,Z 260.318,A -85,B 0,C 180,E1 -20807.698,E2 -20807.698} C_VEL
LIN {X 0,Y 213.758,Z 260.357,A -85,B 0,C 180,E1 -20813.24,E2 -20813.24} C_VEL
LIN {X 0,Y 213.759,Z 260.352,A -85,B 0,C 180,E1 -20817.433,E2 -20817.433} C_VEL
LIN {X 0,Y 213.734,Z 260.351,A -85,B 0,C 180,E1 -20821.746,E2 -20821.746} C_VEL
LIN {X 0,Y 213.719,Z 260.365,A -85,B 0,C 180,E1 -20826.296,E2 -20826.296} C_VEL
LIN {X 0,Y 213.678,Z 260.354,A -85,B 0,C 180,E1 -20831.137,E2 -20831.137} C_VEL
LIN {X 0,Y 213.683,Z 260.366,A -85,B 0,C 180,E1 -20833.688,E2 -20833.688} C_VEL
LIN {X 0,Y 213.685,Z 260.359,A -85,B 0,C 180,E1 -20836.354,E2 -20836.354} C_VEL
LIN {X 0,Y 213.689,Z 260.354,A -85,B 0,C 180,E1 -20841.337,E2 -20841.337} C_VEL
LIN {X 0,Y 213.743,Z 260.356,A -85,B 0,C 180,E1 -20846.026,E2 -20846.026} C_VEL
LIN {X 0,Y 213.737,Z 260.325,A -85,B 0,C 180,E1 -20850.457,E2 -20850.457} C_VEL
LIN {X 0,Y 213.733,Z 260.356,A -85,B 0,C 180,E1 -20854.702,E2 -20854.702} C_VEL
LIN {X 0,Y 213.775,Z 260.352,A -85,B 0,C 180,E1 -20858.808,E2 -20858.808} C_VEL
LIN {X 0,Y 213.884,Z 260.304,A -85,B 0,C 180,E1 -20862.807,E2 -20862.807} C_VEL
LIN {X 0,Y 213.941,Z 260.324,A -85,B 0,C 180,E1 -20866.714,E2 -20866.714} C_VEL
LIN {X 0,Y 214.138,Z 260.309,A -85,B 0,C 180,E1 -20870.563,E2 -20870.563} C_VEL
LIN {X 0,Y 214.078,Z 260.296,A -85,B 0,C 180,E1 -20874.355,E2 -20874.355} C_VEL
LIN {X 0,Y 214.411,Z 260.245,A -85,B 0,C 180,E1 -20878.129,E2 -20878.129} C_VEL
LIN {X 0,Y 214.52,Z 260.249,A -85,B 0,C 180,E1 -20880.007,E2 -20880.007} C_VEL
LIN {X 0,Y 214.411,Z 260.273,A -85,B 0,C 180,E1 -20881.886,E2 -20881.886} C_VEL
LIN {X 0,Y 214.183,Z 260.284,A -85,B 0,C 180,E1 -20887.549,E2 -20887.549} C_VEL
LIN {X 0,Y 214.001,Z 260.307,A -85,B 0,C 180,E1 -20891.371,E2 -20891.371} C_VEL
LIN {X 0,Y 213.915,Z 260.338,A -85,B 0,C 180,E1 -20895.245,E2 -20895.245} C_VEL
LIN {X 0,Y 213.813,Z 260.331,A -85,B 0,C 180,E1 -20899.197,E2 -20899.197} C_VEL
LIN {X 0,Y 213.812,Z 260.344,A -85,B 0,C 180,E1 -20903.238,E2 -20903.238} C_VEL
LIN {X 0,Y 213.805,Z 260.344,A -85,B 0,C 180,E1 -20907.432,E2 -20907.432} C_VEL
LIN {X 0,Y 213.778,Z 260.35,A -85,B 0,C 180,E1 -20911.743,E2 -20911.743} C_VEL
LIN {X 0,Y 213.761,Z 260.344,A -85,B 0,C 180,E1 -20916.292,E2 -20916.292} C_VEL
LIN {X 0,Y 213.716,Z 260.359,A -85,B 0,C 180,E1 -20921.132,E2 -20921.132} C_VEL
LIN {X 0,Y 213.722,Z 260.355,A -85,B 0,C 180,E1 -20923.682,E2 -20923.682} C_VEL
LIN {X 0,Y 213.722,Z 260.357,A -85,B 0,C 180,E1 -20926.348,E2 -20926.348} C_VEL
LIN {X 0,Y 213.688,Z 260.353,A -85,B 0,C 180,E1 -20930.541,E2 -20930.541} C_VEL
LIN {X 0,Y 213.512,Z 260.784,A -85,B 0,C 180,E1 -20931.539,E2 -20931.539} C_VEL
LIN {X 0,Y 212.79,Z 262.74,A -85,B 0,C 180,E1 -20932.955,E2 -20932.955} C_VEL
LIN {X 0,Y 211.963,Z 265.837,A -85,B 0,C 180,E1 -20934.233,E2 -20934.233} C_VEL
LIN {X 0,Y 211.451,Z 269.797,A -85,B 0,C 180,E1 -20935.34,E2 -20935.34} C_VEL
LIN {X 0,Y 211.683,Z 274.436,A -85,B 0,C 180,E1 -20936.213,E2 -20936.213} C_VEL
LIN {X 0,Y 212.515,Z 277.785,A -85,B 0,C 180,E1 -20936.605,E2 -20936.605} C_VEL
LIN {X 0,Y 218.662,Z 294.368,A -85,B 0,C 180,E1 -20938.034,E2 -20938.034} C_VEL
LIN {X 0,Y 219.706,Z 298.436,A -85,B 0,C 180,E1 -20938.314,E2 -20938.314} C_VEL
LIN {X 0,Y 221.941,Z 316.134,A -85,B 0,C 180,E1 -20939.227,E2 -20939.227} C_VEL
LIN {X 0,Y 219.691,Z 375.249,A -85,B 0,C 180,E1 -20941.173,E2 -20941.173} C_VEL
LIN {X 0,Y 218.639,Z 387.591,A -85,B 0,C 180,E1 -20941.89,E2 -20941.89} C_VEL
LIN {X 0,Y 217.266,Z 399.785,A -85,B 0,C 180,E1 -20942.939,E2 -20942.939} C_VEL
LIN {X 0,Y 215.443,Z 412.09,A -85,B 0,C 180,E1 -20944.388,E2 -20944.388} C_VEL
LIN {X 0,Y 213.871,Z 421.117,A -85,B 0,C 180,E1 -20945.744,E2 -20945.744} C_VEL
LIN {X 0,Y 212.046,Z 430.988,A -85,B 0,C 180,E1 -20947.592,E2 -20947.592} C_VEL
LIN {X 0,Y 209.999,Z 441.612,A -85,B 0,C 180,E1 -20950.105,E2 -20950.105} C_VEL
LIN {X 0,Y 208.116,Z 450.681,A -85,B 0,C 180,E1 -20952.81,E2 -20952.81} C_VEL
LIN {X 0,Y 206.493,Z 458.342,A -85,B 0,C 180,E1 -20955.711,E2 -20955.711} C_VEL
LIN {X 0,Y 205.289,Z 465.412,A -85,B 0,C 180,E1 -20959.144,E2 -20959.144} C_VEL
LIN {X 0,Y 204.661,Z 470.068,A -85,B 0,C 180,E1 -20962.102,E2 -20962.102} C_VEL
LIN {X 0,Y 204.422,Z 472.518,A -85,B 0,C 180,E1 -20964.077,E2 -20964.077} C_VEL
LIN {X 0,Y 204.316,Z 474.511,A -85,B 0,C 180,E1 -20966.052,E2 -20966.052} C_VEL
LIN {X 0,Y 204.297,Z 476.081,A -85,B 0,C 180,E1 -20968.026,E2 -20968.026} C_VEL
LIN {X 0,Y 204.367,Z 477.223,A -85,B 0,C 180,E1 -20969.997,E2 -20969.997} C_VEL
LIN {X 0,Y 204.296,Z 477.925,A -85,B 0,C 180,E1 -20971.968,E2 -20971.968} C_VEL
LIN {X 0,Y 204.514,Z 478.183,A -85,B 0,C 180,E1 -20975.914,E2 -20975.914} C_VEL
LIN {X 0,Y 204.782,Z 477.737,A -85,B 0,C 180,E1 -20977.887,E2 -20977.887} C_VEL
LIN {X 0,Y 205.925,Z 475.607,A -85,B 0,C 180,E1 -20981.813,E2 -20981.813} C_VEL
LIN {X 0,Y 207.341,Z 472.96,A -85,B 0,C 180,E1 -20984.724,E2 -20984.724} C_VEL
LIN {X 0,Y 209.242,Z 469.326,A -85,B 0,C 180,E1 -20987.592,E2 -20987.592} C_VEL
LIN {X 0,Y 211.793,Z 464.605,A -85,B 0,C 180,E1 -20990.388,E2 -20990.388} C_VEL
LIN {X 0,Y 214.732,Z 458.666,A -85,B 0,C 180,E1 -20993.122,E2 -20993.122} C_VEL
LIN {X 0,Y 218.018,Z 451.326,A -85,B 0,C 180,E1 -20995.794,E2 -20995.794} C_VEL
LIN {X 0,Y 221.939,Z 442.215,A -85,B 0,C 180,E1 -20998.356,E2 -20998.356} C_VEL
LIN {X 0,Y 225.939,Z 431.731,A -85,B 0,C 180,E1 -21000.617,E2 -21000.617} C_VEL
LIN {X 0,Y 229.449,Z 421.103,A -85,B 0,C 180,E1 -21002.41,E2 -21002.41} C_VEL
LIN {X 0,Y 232.87,Z 409.061,A -85,B 0,C 180,E1 -21003.937,E2 -21003.937} C_VEL
LIN {X 0,Y 235.73,Z 396.268,A -85,B 0,C 180,E1 -21005.151,E2 -21005.151} C_VEL
LIN {X 0,Y 237.807,Z 384.049,A -85,B 0,C 180,E1 -21005.967,E2 -21005.967} C_VEL
LIN {X 0,Y 239.249,Z 370.929,A -85,B 0,C 180,E1 -21006.533,E2 -21006.533} C_VEL
LIN {X 0,Y 241.906,Z 323.987,A -85,B 0,C 180,E1 -21007.933,E2 -21007.933} C_VEL
LIN {X 0,Y 236.938,Z 312.483,A -85,B 0,C 180,E1 -21009.656,E2 -21009.656} C_VEL
LIN {X 0,Y 230.837,Z 300.214,A -85,B 0,C 180,E1 -21011.89,E2 -21011.89} C_VEL
LIN {X 0,Y 225.174,Z 290.455,A -85,B 0,C 180,E1 -21014.114,E2 -21014.114} C_VEL
LIN {X 0,Y 221.805,Z 285.101,A -85,B 0,C 180,E1 -21015.521,E2 -21015.521} C_VEL
LIN {X 0,Y 219.361,Z 281.36,A -85,B 0,C 180,E1 -21016.594,E2 -21016.594} C_VEL
LIN {X 0,Y 215.951,Z 276.325,A -85,B 0,C 180,E1 -21018.187,E2 -21018.187} C_VEL
LIN {X 0,Y 211.768,Z 270.591,A -85,B 0,C 180,E1 -21020.308,E2 -21020.308} C_VEL
LIN {X 0,Y 207.997,Z 265.21,A -85,B 0,C 180,E1 -21022.533,E2 -21022.533} C_VEL
LIN {X 0,Y 206.798,Z 261.648,A -85,B 0,C 180,E1 -21025.885,E2 -21025.885} C_VEL
LIN {X 0,Y 206.696,Z 261.228,A -85,B 0,C 180,E1 -21027.034,E2 -21027.034} C_VEL
LIN {X 0,Y 206.707,Z 261.232,A -85,B 0,C 180,E1 -21032.12,E2 -21032.12} C_VEL
LIN {X 0,Y 206.725,Z 261.235,A -85,B 0,C 180,E1 -21036.614,E2 -21036.614} C_VEL
LIN {X 0,Y 206.817,Z 261.213,A -85,B 0,C 180,E1 -21042.184,E2 -21042.184} C_VEL
LIN {X 0,Y 206.867,Z 261.211,A -85,B 0,C 180,E1 -21046.235,E2 -21046.235} C_VEL
LIN {X 0,Y 207.071,Z 261.192,A -85,B 0,C 180,E1 -21050.222,E2 -21050.222} C_VEL
LIN {X 0,Y 207.026,Z 261.193,A -85,B 0,C 180,E1 -21054.147,E2 -21054.147} C_VEL
LIN {X 0,Y 207.33,Z 261.149,A -85,B 0,C 180,E1 -21058.05,E2 -21058.05} C_VEL
LIN {X 0,Y 207.466,Z 261.135,A -85,B 0,C 180,E1 -21059.992,E2 -21059.992} C_VEL
LIN {X 0,Y 207.331,Z 261.146,A -85,B 0,C 180,E1 -21061.935,E2 -21061.935} C_VEL
LIN {X 0,Y 207.108,Z 261.187,A -85,B 0,C 180,E1 -21067.793,E2 -21067.793} C_VEL
LIN {X 0,Y 206.898,Z 261.211,A -85,B 0,C 180,E1 -21071.752,E2 -21071.752} C_VEL
LIN {X 0,Y 206.889,Z 261.449,A -85,B 0,C 180,E1 -21075.256,E2 -21075.256} C_VEL
LIN {X 0,Y 207.204,Z 262.798,A -85,B 0,C 180,E1 -21076.178,E2 -21076.178} C_VEL
LIN {X 0,Y 208.82,Z 265.327,A -85,B 0,C 180,E1 -21077.21,E2 -21077.21} C_VEL
LIN {X 0,Y 211.891,Z 268.737,A -85,B 0,C 180,E1 -21078.859,E2 -21078.859} C_VEL
LIN {X 0,Y 216.36,Z 274.735,A -85,B 0,C 180,E1 -21081.114,E2 -21081.114} C_VEL
LIN {X 0,Y 220.611,Z 280.75,A -85,B 0,C 180,E1 -21083.058,E2 -21083.058} C_VEL
LIN {X 0,Y 225.76,Z 288.603,A -85,B 0,C 180,E1 -21085.214,E2 -21085.214} C_VEL
LIN {X 0,Y 232.916,Z 300.953,A -85,B 0,C 180,E1 -21087.975,E2 -21087.975} C_VEL
LIN {X 0,Y 238.94,Z 312.889,A -85,B 0,C 180,E1 -21090.103,E2 -21090.103} C_VEL
LIN {X 0,Y 242.068,Z 320.027,A -85,B 0,C 180,E1 -21091.171,E2 -21091.171} C_VEL
LIN {X 0,Y 239.8,Z 360.519,A -85,B 0,C 180,E1 -21092.369,E2 -21092.369} C_VEL
LIN {X 0,Y 238.65,Z 374.179,A -85,B 0,C 180,E1 -21092.854,E2 -21092.854} C_VEL
LIN {X 0,Y 236.82,Z 387.13,A -85,B 0,C 180,E1 -21093.63,E2 -21093.63} C_VEL
LIN {X 0,Y 234.257,Z 400.058,A -85,B 0,C 180,E1 -21094.742,E2 -21094.742} C_VEL
LIN {X 0,Y 231.431,Z 411.291,A -85,B 0,C 180,E1 -21096.052,E2 -21096.052} C_VEL
LIN {X 0,Y 227.953,Z 422.632,A -85,B 0,C 180,E1 -21097.785,E2 -21097.785} C_VEL
LIN {X 0,Y 224.211,Z 433.079,A -85,B 0,C 180,E1 -21099.834,E2 -21099.834} C_VEL
LIN {X 0,Y 220.433,Z 442.231,A -85,B 0,C 180,E1 -21102.138,E2 -21102.138} C_VEL
LIN {X 0,Y 217.013,Z 449.806,A -85,B 0,C 180,E1 -21104.568,E2 -21104.568} C_VEL
LIN {X 0,Y 213.518,Z 457.069,A -85,B 0,C 180,E1 -21107.569,E2 -21107.569} C_VEL
LIN {X 0,Y 210.602,Z 462.733,A -85,B 0,C 180,E1 -21110.655,E2 -21110.655} C_VEL
LIN {X 0,Y 208.043,Z 467.36,A -85,B 0,C 180,E1 -21114.154,E2 -21114.154} C_VEL
LIN {X 0,Y 206.532,Z 470,A -85,B 0,C 180,E1 -21117.016,E2 -21117.016} C_VEL
LIN {X 0,Y 205.597,Z 471.376,A -85,B 0,C 180,E1 -21119.157,E2 -21119.157} C_VEL
LIN {X 0,Y 204.896,Z 472.279,A -85,B 0,C 180,E1 -21121.305,E2 -21121.305} C_VEL
LIN {X 0,Y 204.419,Z 472.672,A -85,B 0,C 180,E1 -21123.456,E2 -21123.456} C_VEL
LIN {X 0,Y 204.022,Z 472.632,A -85,B 0,C 180,E1 -21125.587,E2 -21125.587} C_VEL
LIN {X 0,Y 203.856,Z 471.8,A -85,B 0,C 180,E1 -21128.538,E2 -21128.538} C_VEL
LIN {X 0,Y 203.932,Z 469.748,A -85,B 0,C 180,E1 -21131.934,E2 -21131.934} C_VEL
LIN {X 0,Y 204.246,Z 467.429,A -85,B 0,C 180,E1 -21134.428,E2 -21134.428} C_VEL
LIN {X 0,Y 204.791,Z 464.131,A -85,B 0,C 180,E1 -21137.114,E2 -21137.114} C_VEL
LIN {X 0,Y 205.63,Z 459.215,A -85,B 0,C 180,E1 -21140.164,E2 -21140.164} C_VEL
LIN {X 0,Y 206.701,Z 453.003,A -85,B 0,C 180,E1 -21143.169,E2 -21143.169} C_VEL
LIN {X 0,Y 208.329,Z 445.23,A -85,B 0,C 180,E1 -21146.134,E2 -21146.134} C_VEL
LIN {X 0,Y 209.972,Z 437.129,A -85,B 0,C 180,E1 -21148.605,E2 -21148.605} C_VEL
LIN {X 0,Y 211.969,Z 427.488,A -85,B 0,C 180,E1 -21150.953,E2 -21150.953} C_VEL
LIN {X 0,Y 214.042,Z 416.598,A -85,B 0,C 180,E1 -21153.061,E2 -21153.061} C_VEL
LIN {X 0,Y 215.761,Z 406.085,A -85,B 0,C 180,E1 -21154.674,E2 -21154.674} C_VEL
LIN {X 0,Y 217.385,Z 394.59,A -85,B 0,C 180,E1 -21156.034,E2 -21156.034} C_VEL
LIN {X 0,Y 218.779,Z 381.66,A -85,B 0,C 180,E1 -21157.154,E2 -21157.154} C_VEL
LIN {X 0,Y 219.809,Z 368.111,A -85,B 0,C 180,E1 -21157.929,E2 -21157.929} C_VEL
LIN {X 0,Y 222.279,Z 304.168,A -85,B 0,C 180,E1 -21159.994,E2 -21159.994} C_VEL
LIN {X 0,Y 221.292,Z 298.828,A -85,B 0,C 180,E1 -21160.306,E2 -21160.306} C_VEL
LIN {X 0,Y 214.811,Z 279.928,A -85,B 0,C 180,E1 -21161.831,E2 -21161.831} C_VEL
LIN {X 0,Y 208.039,Z 264.319,A -85,B 0,C 180,E1 -21163.373,E2 -21163.373} C_VEL
LIN {X 0,Y 206.958,Z 261.849,A -85,B 0,C 180,E1 -21163.754,E2 -21163.754} C_VEL
LIN {X 0,Y 206.847,Z 261.259,A -85,B 0,C 180,E1 -21164.264,E2 -21164.264} C_VEL
LIN {X 0,Y 206.827,Z 261.2,A -85,B 0,C 180,E1 -21167.96,E2 -21167.96} C_VEL
LIN {X 0,Y 206.701,Z 261.237,A -85,B 0,C 180,E1 -21173.386,E2 -21173.386} C_VEL
LIN {X 0,Y 206.661,Z 261.243,A -85,B 0,C 180,E1 -21178.434,E2 -21178.434} C_VEL
LIN {X 0,Y 206.67,Z 261.228,A -85,B 0,C 180,E1 -21182.966,E2 -21182.966} C_VEL
LIN {X 0,Y 206.646,Z 261.237,A -85,B 0,C 180,E1 -21187.75,E2 -21187.75} C_VEL
LIN {X 0,Y 206.611,Z 261.238,A -85,B 0,C 180,E1 -21191.567,E2 -21191.567} C_VEL
LIN {X 0,Y 206.613,Z 261.245,A -85,B 0,C 180,E1 -21195.591,E2 -21195.591} C_VEL
LIN {X 0,Y 206.632,Z 261.22,A -85,B 0,C 180,E1 -21199.754,E2 -21199.754} C_VEL
LIN {X 0,Y 206.689,Z 261.24,A -85,B 0,C 180,E1 -21204.698,E2 -21204.698} C_VEL
LIN {X 0,Y 206.685,Z 261.205,A -85,B 0,C 180,E1 -21209.343,E2 -21209.343} C_VEL
LIN {X 0,Y 206.666,Z 261.232,A -85,B 0,C 180,E1 -21213.772,E2 -21213.772} C_VEL
LIN {X 0,Y 206.711,Z 261.232,A -85,B 0,C 180,E1 -21218.047,E2 -21218.047} C_VEL
LIN {X 0,Y 206.822,Z 261.185,A -85,B 0,C 180,E1 -21222.201,E2 -21222.201} C_VEL
LIN {X 0,Y 206.88,Z 261.197,A -85,B 0,C 180,E1 -21226.252,E2 -21226.252} C_VEL
LIN {X 0,Y 207.082,Z 261.189,A -85,B 0,C 180,E1 -21230.238,E2 -21230.238} C_VEL
LIN {X 0,Y 207.041,Z 261.172,A -85,B 0,C 180,E1 -21234.163,E2 -21234.163} C_VEL
LIN {X 0,Y 207.35,Z 261.122,A -85,B 0,C 180,E1 -21238.065,E2 -21238.065} C_VEL
LIN {X 0,Y 207.488,Z 261.125,A -85,B 0,C 180,E1 -21240.008,E2 -21240.008} C_VEL
LIN {X 0,Y 207.351,Z 261.153,A -85,B 0,C 180,E1 -21241.95,E2 -21241.95} C_VEL
LIN {X 0,Y 207.129,Z 261.157,A -85,B 0,C 180,E1 -21247.808,E2 -21247.808} C_VEL
LIN {X 0,Y 206.925,Z 261.193,A -85,B 0,C 180,E1 -21251.766,E2 -21251.766} C_VEL
LIN {X 0,Y 206.842,Z 261.219,A -85,B 0,C 180,E1 -21255.78,E2 -21255.78} C_VEL
LIN {X 0,Y 206.732,Z 261.208,A -85,B 0,C 180,E1 -21259.881,E2 -21259.881} C_VEL
LIN {X 0,Y 206.752,Z 261.228,A -85,B 0,C 180,E1 -21264.081,E2 -21264.081} C_VEL
LIN {X 0,Y 206.707,Z 261.221,A -85,B 0,C 180,E1 -21268.432,E2 -21268.432} C_VEL
LIN {X 0,Y 206.714,Z 261.235,A -85,B 0,C 180,E1 -21272.962,E2 -21272.962} C_VEL
LIN {X 0,Y 206.72,Z 261.226,A -85,B 0,C 180,E1 -21275.315,E2 -21275.315} C_VEL
LIN {X 0,Y 206.665,Z 261.241,A -85,B 0,C 180,E1 -21280.258,E2 -21280.258} C_VEL
LIN {X 0,Y 206.651,Z 261.244,A -85,B 0,C 180,E1 -21284.419,E2 -21284.419} C_VEL
LIN {X 0,Y 206.652,Z 261.24,A -85,B 0,C 180,E1 -21288.443,E2 -21288.443} C_VEL
LIN {X 0,Y 206.761,Z 261.315,A -85,B 0,C 180,E1 -21292.861,E2 -21292.861} C_VEL
LIN {X 0,Y 207.929,Z 266.359,A -85,B 0,C 180,E1 -21295.417,E2 -21295.417} C_VEL
LIN {X 0,Y 209.742,Z 271.1,A -85,B 0,C 180,E1 -21295.97,E2 -21295.97} C_VEL
LIN {X 0,Y 212.515,Z 277.785,A -85,B 0,C 180,E1 -21296.605,E2 -21296.605} C_VEL
LIN {X 0,Y 213.845,Z 283.383,A -85,B 0,C 180,E1 -21297,E2 -21297} C_VEL
LIN {X 0,Y 214.381,Z 293.181,A -85,B 0,C 180,E1 -21297.444,E2 -21297.444} C_VEL
LIN {X 0,Y 214.234,Z 301.196,A -85,B 0,C 180,E1 -21297.73,E2 -21297.73} C_VEL
LIN {X 0,Y 214.522,Z 309.158,A -85,B 0,C 180,E1 -21298.069,E2 -21298.069} C_VEL
LIN {X 0,Y 215.459,Z 317.156,A -85,B 0,C 180,E1 -21298.487,E2 -21298.487} C_VEL
LIN {X 0,Y 213.193,Z 374.749,A -85,B 0,C 180,E1 -21300.429,E2 -21300.429} C_VEL
LIN {X 0,Y 212.036,Z 387.776,A -85,B 0,C 180,E1 -21301.204,E2 -21301.204} C_VEL
LIN {X 0,Y 210.616,Z 399.898,A -85,B 0,C 180,E1 -21302.282,E2 -21302.282} C_VEL
LIN {X 0,Y 208.735,Z 412.142,A -85,B 0,C 180,E1 -21303.771,E2 -21303.771} C_VEL
LIN {X 0,Y 207.112,Z 421.146,A -85,B 0,C 180,E1 -21305.167,E2 -21305.167} C_VEL
LIN {X 0,Y 205.223,Z 430.993,A -85,B 0,C 180,E1 -21307.071,E2 -21307.071} C_VEL
LIN {X 0,Y 203.267,Z 440.511,A -85,B 0,C 180,E1 -21309.365,E2 -21309.365} C_VEL
LIN {X 0,Y 201.55,Z 448.409,A -85,B 0,C 180,E1 -21311.707,E2 -21311.707} C_VEL
LIN {X 0,Y 199.813,Z 456.548,A -85,B 0,C 180,E1 -21314.701,E2 -21314.701} C_VEL
LIN {X 0,Y 198.601,Z 463.063,A -85,B 0,C 180,E1 -21317.738,E2 -21317.738} C_VEL
LIN {X 0,Y 197.808,Z 468.207,A -85,B 0,C 180,E1 -21320.797,E2 -21320.797} C_VEL
LIN {X 0,Y 197.361,Z 472.177,A -85,B 0,C 180,E1 -21323.864,E2 -21323.864} C_VEL
LIN {X 0,Y 197.199,Z 474.613,A -85,B 0,C 180,E1 -21326.372,E2 -21326.372} C_VEL
LIN {X 0,Y 197.273,Z 477.019,A -85,B 0,C 180,E1 -21329.997,E2 -21329.997} C_VEL
LIN {X 0,Y 197.195,Z 478.093,A -85,B 0,C 180,E1 -21333.614,E2 -21333.614} C_VEL
LIN {X 0,Y 197.43,Z 478.102,A -85,B 0,C 180,E1 -21336.127,E2 -21336.127} C_VEL
LIN {X 0,Y 197.736,Z 477.699,A -85,B 0,C 180,E1 -21338.17,E2 -21338.17} C_VEL
LIN {X 0,Y 198.249,Z 476.894,A -85,B 0,C 180,E1 -21340.206,E2 -21340.206} C_VEL
LIN {X 0,Y 199.921,Z 474.056,A -85,B 0,C 180,E1 -21344.242,E2 -21344.242} C_VEL
LIN {X 0,Y 201.737,Z 470.84,A -85,B 0,C 180,E1 -21347.221,E2 -21347.221} C_VEL
LIN {X 0,Y 204.205,Z 466.589,A -85,B 0,C 180,E1 -21350.127,E2 -21350.127} C_VEL
LIN {X 0,Y 207.724,Z 460.189,A -85,B 0,C 180,E1 -21353.421,E2 -21353.421} C_VEL
LIN {X 0,Y 211.05,Z 453.233,A -85,B 0,C 180,E1 -21356.179,E2 -21356.179} C_VEL
LIN {X 0,Y 215.06,Z 444.556,A -85,B 0,C 180,E1 -21358.814,E2 -21358.814} C_VEL
LIN {X 0,Y 218.76,Z 435.7,A -85,B 0,C 180,E1 -21360.929,E2 -21360.929} C_VEL
LIN {X 0,Y 222.723,Z 424.803,A -85,B 0,C 180,E1 -21362.975,E2 -21362.975} C_VEL
LIN {X 0,Y 226.201,Z 413.798,A -85,B 0,C 180,E1 -21364.539,E2 -21364.539} C_VEL
LIN {X 0,Y 229.355,Z 401.526,A -85,B 0,C 180,E1 -21365.872,E2 -21365.872} C_VEL
LIN {X 0,Y 231.691,Z 389.893,A -85,B 0,C 180,E1 -21366.801,E2 -21366.801} C_VEL
LIN {X 0,Y 233.554,Z 376.799,A -85,B 0,C 180,E1 -21367.509,E2 -21367.509} C_VEL
LIN {X 0,Y 234.926,Z 358.601,A -85,B 0,C 180,E1 -21368.102,E2 -21368.102} C_VEL
LIN {X 0,Y 236.785,Z 326.275,A -85,B 0,C 180,E1 -21369.077,E2 -21369.077} C_VEL
LIN {X 0,Y 231.22,Z 313.545,A -85,B 0,C 180,E1 -21371.134,E2 -21371.134} C_VEL
LIN {X 0,Y 226.177,Z 303.473,A -85,B 0,C 180,E1 -21373.122,E2 -21373.122} C_VEL
LIN {X 0,Y 221.291,Z 294.99,A -85,B 0,C 180,E1 -21375.155,E2 -21375.155} C_VEL
LIN {X 0,Y 216.502,Z 287.258,A -85,B 0,C 180,E1 -21377.311,E2 -21377.311} C_VEL
LIN {X 0,Y 212.929,Z 281.911,A -85,B 0,C 180,E1 -21379.074,E2 -21379.074} C_VEL
LIN {X 0,Y 208.999,Z 276.391,A -85,B 0,C 180,E1 -21381.168,E2 -21381.168} C_VEL
LIN {X 0,Y 204.65,Z 270.385,A -85,B 0,C 180,E1 -21383.749,E2 -21383.749} C_VEL
LIN {X 0,Y 201.739,Z 266.877,A -85,B 0,C 180,E1 -21385.664,E2 -21385.664} C_VEL
LIN {X 0,Y 200.552,Z 264.802,A -85,B 0,C 180,E1 -21386.765,E2 -21386.765} C_VEL
LIN {X 0,Y 199.632,Z 262.172,A -85,B 0,C 180,E1 -21390.027,E2 -21390.027} C_VEL
LIN {X 0,Y 199.635,Z 262.119,A -85,B 0,C 180,E1 -21392.756,E2 -21392.756} C_VEL
LIN {X 0,Y 199.669,Z 262.111,A -85,B 0,C 180,E1 -21397.213,E2 -21397.213} C_VEL
LIN {X 0,Y 199.741,Z 262.098,A -85,B 0,C 180,E1 -21401.795,E2 -21401.795} C_VEL
LIN {X 0,Y 199.805,Z 262.097,A -85,B 0,C 180,E1 -21405.739,E2 -21405.739} C_VEL
LIN {X 0,Y 200.015,Z 262.07,A -85,B 0,C 180,E1 -21409.874,E2 -21409.874} C_VEL
LIN {X 0,Y 199.99,Z 262.066,A -85,B 0,C 180,E1 -21413.941,E2 -21413.941} C_VEL
LIN {X 0,Y 200.272,Z 262.027,A -85,B 0,C 180,E1 -21417.981,E2 -21417.981} C_VEL
LIN {X 0,Y 200.433,Z 262.01,A -85,B 0,C 180,E1 -21419.992,E2 -21419.992} C_VEL
LIN {X 0,Y 199.975,Z 262.071,A -85,B 0,C 180,E1 -21424.023,E2 -21424.023} C_VEL
LIN {X 0,Y 200.056,Z 262.061,A -85,B 0,C 180,E1 -21428.07,E2 -21428.07} C_VEL
LIN {X 0,Y 199.908,Z 262.293,A -85,B 0,C 180,E1 -21431.718,E2 -21431.718} C_VEL
LIN {X 0,Y 200.223,Z 263.671,A -85,B 0,C 180,E1 -21432.342,E2 -21432.342} C_VEL
LIN {X 0,Y 201.514,Z 265.867,A -85,B 0,C 180,E1 -21433.351,E2 -21433.351} C_VEL
LIN {X 0,Y 204.383,Z 268.343,A -85,B 0,C 180,E1 -21435.191,E2 -21435.191} C_VEL
LIN {X 0,Y 206.643,Z 271.721,A -85,B 0,C 180,E1 -21436.607,E2 -21436.607} C_VEL
LIN {X 0,Y 209.445,Z 274.963,A -85,B 0,C 180,E1 -21438.177,E2 -21438.177} C_VEL
LIN {X 0,Y 213.762,Z 280.925,A -85,B 0,C 180,E1 -21440.445,E2 -21440.445} C_VEL
LIN {X 0,Y 218.064,Z 287.215,A -85,B 0,C 180,E1 -21442.509,E2 -21442.509} C_VEL
LIN {X 0,Y 222.871,Z 294.886,A -85,B 0,C 180,E1 -21444.607,E2 -21444.607} C_VEL
LIN {X 0,Y 229.357,Z 306.35,A -85,B 0,C 180,E1 -21447.216,E2 -21447.216} C_VEL
LIN {X 0,Y 234.933,Z 317.799,A -85,B 0,C 180,E1 -21449.306,E2 -21449.306} C_VEL
LIN {X 0,Y 237.027,Z 322.793,A -85,B 0,C 180,E1 -21450.066,E2 -21450.066} C_VEL
LIN {X 0,Y 233.964,Z 370.279,A -85,B 0,C 180,E1 -21451.496,E2 -21451.496} C_VEL
LIN {X 0,Y 232.132,Z 384.218,A -85,B 0,C 180,E1 -21452.232,E2 -21452.232} C_VEL
LIN {X 0,Y 229.779,Z 396.578,A -85,B 0,C 180,E1 -21453.217,E2 -21453.217} C_VEL
LIN {X 0,Y 226.943,Z 408.052,A -85,B 0,C 180,E1 -21454.465,E2 -21454.465} C_VEL
LIN {X 0,Y 223.311,Z 420.075,A -85,B 0,C 180,E1 -21456.189,E2 -21456.189} C_VEL
LIN {X 0,Y 219.717,Z 430.02,A -85,B 0,C 180,E1 -21458.037,E2 -21458.037} C_VEL
LIN {X 0,Y 216.075,Z 438.845,A -85,B 0,C 180,E1 -21460.11,E2 -21460.11} C_VEL
LIN {X 0,Y 212.296,Z 447.099,A -85,B 0,C 180,E1 -21462.564,E2 -21462.564} C_VEL
LIN {X 0,Y 208.384,Z 454.977,A -85,B 0,C 180,E1 -21465.592,E2 -21465.592} C_VEL
LIN {X 0,Y 204.781,Z 461.573,A -85,B 0,C 180,E1 -21469.014,E2 -21469.014} C_VEL
LIN {X 0,Y 201.948,Z 466.452,A -85,B 0,C 180,E1 -21472.479,E2 -21472.479} C_VEL
LIN {X 0,Y 199.985,Z 469.689,A -85,B 0,C 180,E1 -21475.79,E2 -21475.79} C_VEL
LIN {X 0,Y 198.946,Z 471.167,A -85,B 0,C 180,E1 -21478.006,E2 -21478.006} C_VEL
LIN {X 0,Y 198.09,Z 472.182,A -85,B 0,C 180,E1 -21480.222,E2 -21480.222} C_VEL
LIN {X 0,Y 197.421,Z 472.761,A -85,B 0,C 180,E1 -21482.848,E2 -21482.848} C_VEL
LIN {X 0,Y 196.786,Z 472.399,A -85,B 0,C 180,E1 -21486.872,E2 -21486.872} C_VEL
LIN {X 0,Y 196.744,Z 471.565,A -85,B 0,C 180,E1 -21489.074,E2 -21489.074} C_VEL
LIN {X 0,Y 196.768,Z 470.245,A -85,B 0,C 180,E1 -21491.253,E2 -21491.253} C_VEL
LIN {X 0,Y 197.129,Z 467.684,A -85,B 0,C 180,E1 -21494.243,E2 -21494.243} C_VEL
LIN {X 0,Y 197.81,Z 463.494,A -85,B 0,C 180,E1 -21497.695,E2 -21497.695} C_VEL
LIN {X 0,Y 198.73,Z 458.46,A -85,B 0,C 180,E1 -21500.804,E2 -21500.804} C_VEL
LIN {X 0,Y 199.958,Z 451.952,A -85,B 0,C 180,E1 -21503.951,E2 -21503.951} C_VEL
LIN {X 0,Y 201.628,Z 443.867,A -85,B 0,C 180,E1 -21507.006,E2 -21507.006} C_VEL
LIN {X 0,Y 203.453,Z 435.39,A -85,B 0,C 180,E1 -21509.558,E2 -21509.558} C_VEL
LIN {X 0,Y 205.561,Z 425.423,A -85,B 0,C 180,E1 -21511.962,E2 -21511.962} C_VEL
LIN {X 0,Y 207.544,Z 415.384,A -85,B 0,C 180,E1 -21513.886,E2 -21513.886} C_VEL
LIN {X 0,Y 209.347,Z 404.473,A -85,B 0,C 180,E1 -21515.542,E2 -21515.542} C_VEL
LIN {X 0,Y 211.064,Z 392.433,A -85,B 0,C 180,E1 -21516.936,E2 -21516.936} C_VEL
LIN {X 0,Y 212.431,Z 379.444,A -85,B 0,C 180,E1 -21518.031,E2 -21518.031} C_VEL
LIN {X 0,Y 213.352,Z 366.858,A -85,B 0,C 180,E1 -21518.708,E2 -21518.708} C_VEL
LIN {X 0,Y 215.827,Z 304.957,A -85,B 0,C 180,E1 -21520.753,E2 -21520.753} C_VEL
LIN {X 0,Y 215.05,Z 301.058,A -85,B 0,C 180,E1 -21520.999,E2 -21520.999} C_VEL
LIN {X 0,Y 209.105,Z 283.415,A -85,B 0,C 180,E1 -21522.473,E2 -21522.473} C_VEL
LIN {X 0,Y 202.421,Z 267.973,A -85,B 0,C 180,E1 -21524.047,E2 -21524.047} C_VEL
LIN {X 0,Y 199.993,Z 263.028,A -85,B 0,C 180,E1 -21524.698,E2 -21524.698} C_VEL
LIN {X 0,Y 199.809,Z 262.172,A -85,B 0,C 180,E1 -21525.103,E2 -21525.103} C_VEL
LIN {X 0,Y 199.753,Z 262.086,A -85,B 0,C 180,E1 -21528.464,E2 -21528.464} C_VEL
LIN {X 0,Y 199.666,Z 262.115,A -85,B 0,C 180,E1 -21533.795,E2 -21533.795} C_VEL
LIN {X 0,Y 199.638,Z 262.117,A -85,B 0,C 180,E1 -21538.367,E2 -21538.367} C_VEL
LIN {X 0,Y 199.641,Z 262.102,A -85,B 0,C 180,E1 -21542.359,E2 -21542.359} C_VEL
LIN {X 0,Y 199.595,Z 262.121,A -85,B 0,C 180,E1 -21546.773,E2 -21546.773} C_VEL
LIN {X 0,Y 199.574,Z 262.104,A -85,B 0,C 180,E1 -21549.34,E2 -21549.34} C_VEL
LIN {X 0,Y 199.547,Z 262.121,A -85,B 0,C 180,E1 -21552.315,E2 -21552.315} C_VEL
LIN {X 0,Y 199.559,Z 262.124,A -85,B 0,C 180,E1 -21555.236,E2 -21555.236} C_VEL
LIN {X 0,Y 199.554,Z 262.103,A -85,B 0,C 180,E1 -21558.011,E2 -21558.011} C_VEL
LIN {X 0,Y 199.583,Z 262.104,A -85,B 0,C 180,E1 -21560.782,E2 -21560.782} C_VEL
LIN {X 0,Y 199.6,Z 262.118,A -85,B 0,C 180,E1 -21565.722,E2 -21565.722} C_VEL
LIN {X 0,Y 199.676,Z 262.09,A -85,B 0,C 180,E1 -21568.143,E2 -21568.143} C_VEL
LIN {X 0,Y 199.616,Z 262.101,A -85,B 0,C 180,E1 -21572.771,E2 -21572.771} C_VEL
LIN {X 0,Y 199.667,Z 262.114,A -85,B 0,C 180,E1 -21577.23,E2 -21577.23} C_VEL
LIN {X 0,Y 199.745,Z 262.068,A -85,B 0,C 180,E1 -21581.812,E2 -21581.812} C_VEL
LIN {X 0,Y 199.816,Z 262.071,A -85,B 0,C 180,E1 -21585.755,E2 -21585.755} C_VEL
LIN {X 0,Y 200.027,Z 262.07,A -85,B 0,C 180,E1 -21589.89,E2 -21589.89} C_VEL
LIN {X 0,Y 200.005,Z 262.049,A -85,B 0,C 180,E1 -21593.957,E2 -21593.957} C_VEL
LIN {X 0,Y 200.292,Z 261.999,A -85,B 0,C 180,E1 -21597.997,E2 -21597.997} C_VEL
LIN {X 0,Y 200.455,Z 262,A -85,B 0,C 180,E1 -21600.008,E2 -21600.008} C_VEL
LIN {X 0,Y 199.992,Z 262.074,A -85,B 0,C 180,E1 -21604.038,E2 -21604.038} C_VEL
LIN {X 0,Y 200.078,Z 262.03,A -85,B 0,C 180,E1 -21608.085,E2 -21608.085} C_VEL
LIN {X 0,Y 199.876,Z 262.072,A -85,B 0,C 180,E1 -21612.187,E2 -21612.187} C_VEL
LIN {X 0,Y 199.779,Z 262.099,A -85,B 0,C 180,E1 -21616.353,E2 -21616.353} C_VEL
LIN {X 0,Y 199.665,Z 262.085,A -85,B 0,C 180,E1 -21620.617,E2 -21620.617} C_VEL
LIN {X 0,Y 199.667,Z 262.115,A -85,B 0,C 180,E1 -21624.993,E2 -21624.993} C_VEL
LIN {X 0,Y 199.628,Z 262.097,A -85,B 0,C 180,E1 -21629.538,E2 -21629.538} C_VEL
LIN {X 0,Y 199.685,Z 262.108,A -85,B 0,C 180,E1 -21632.356,E2 -21632.356} C_VEL
LIN {X 0,Y 199.635,Z 262.101,A -85,B 0,C 180,E1 -21636.769,E2 -21636.769} C_VEL
LIN {X 0,Y 199.614,Z 262.119,A -85,B 0,C 180,E1 -21639.335,E2 -21639.335} C_VEL
LIN {X 0,Y 199.585,Z 262.11,A -85,B 0,C 180,E1 -21642.309,E2 -21642.309} C_VEL
LIN {X 0,Y 199.597,Z 262.124,A -85,B 0,C 180,E1 -21645.23,E2 -21645.23} C_VEL
LIN {X 0,Y 199.591,Z 262.116,A -85,B 0,C 180,E1 -21648.004,E2 -21648.004} C_VEL
LIN {X 0,Y 199.684,Z 262.186,A -85,B 0,C 180,E1 -21652.137,E2 -21652.137} C_VEL
LIN {X 0,Y 200.44,Z 265.506,A -85,B 0,C 180,E1 -21653.992,E2 -21653.992} C_VEL
LIN {X 0,Y 200.863,Z 266.973,A -85,B 0,C 180,E1 -21654.457,E2 -21654.457} C_VEL
LIN {X 0,Y 208.116,Z 284.52,A -85,B 0,C 180,E1 -21656.271,E2 -21656.271} C_VEL
LIN {X 0,Y 213.31,Z 299.52,A -85,B 0,C 180,E1 -21657.546,E2 -21657.546} C_VEL
LIN {X 0,Y 214.522,Z 309.158,A -85,B 0,C 180,E1 -21658.069,E2 -21658.069} C_VEL
LIN {X 0,Y 214.235,Z 313.064,A -85,B 0,C 180,E1 -21658.18,E2 -21658.18} C_VEL
LIN {X 0,Y 211.939,Z 319.35,A -85,B 0,C 180,E1 -21658.127,E2 -21658.127} C_VEL
LIN {X 0,Y 209.335,Z 325.653,A -85,B 0,C 180,E1 -21658.034,E2 -21658.034} C_VEL
LIN {X 0,Y 208.6,Z 329.617,A -85,B 0,C 180,E1 -21658.092,E2 -21658.092} C_VEL
LIN {X 0,Y 206.662,Z 375.074,A -85,B 0,C 180,E1 -21659.679,E2 -21659.679} C_VEL
LIN {X 0,Y 205.464,Z 387.961,A -85,B 0,C 180,E1 -21660.474,E2 -21660.474} C_VEL
LIN {X 0,Y 203.995,Z 400.01,A -85,B 0,C 180,E1 -21661.581,E2 -21661.581} C_VEL
LIN {X 0,Y 202.053,Z 412.193,A -85,B 0,C 180,E1 -21663.113,E2 -21663.113} C_VEL
LIN {X 0,Y 200.376,Z 421.174,A -85,B 0,C 180,E1 -21664.551,E2 -21664.551} C_VEL
LIN {X 0,Y 198.417,Z 430.997,A -85,B 0,C 180,E1 -21666.514,E2 -21666.514} C_VEL
LIN {X 0,Y 196.294,Z 440.978,A -85,B 0,C 180,E1 -21669.017,E2 -21669.017} C_VEL
LIN {X 0,Y 194.437,Z 449.136,A -85,B 0,C 180,E1 -21671.559,E2 -21671.559} C_VEL
LIN {X 0,Y 192.669,Z 457.118,A -85,B 0,C 180,E1 -21674.662,E2 -21674.662} C_VEL
LIN {X 0,Y 191.644,Z 462.518,A -85,B 0,C 180,E1 -21677.286,E2 -21677.286} C_VEL
LIN {X 0,Y 190.772,Z 467.77,A -85,B 0,C 180,E1 -21680.454,E2 -21680.454} C_VEL
LIN {X 0,Y 190.299,Z 471.825,A -85,B 0,C 180,E1 -21683.636,E2 -21683.636} C_VEL
LIN {X 0,Y 190.109,Z 474.623,A -85,B 0,C 180,E1 -21686.605,E2 -21686.605} C_VEL
LIN {X 0,Y 190.181,Z 476.794,A -85,B 0,C 180,E1 -21689.997,E2 -21689.997} C_VEL
LIN {X 0,Y 190.087,Z 477.873,A -85,B 0,C 180,E1 -21693.282,E2 -21693.282} C_VEL
LIN {X 0,Y 190.375,Z 478.021,A -85,B 0,C 180,E1 -21696.355,E2 -21696.355} C_VEL
LIN {X 0,Y 191.261,Z 476.914,A -85,B 0,C 180,E1 -21700.584,E2 -21700.584} C_VEL
LIN {X 0,Y 193.035,Z 474.178,A -85,B 0,C 180,E1 -21704.762,E2 -21704.762} C_VEL
LIN {X 0,Y 194.953,Z 471.049,A -85,B 0,C 180,E1 -21707.84,E2 -21707.84} C_VEL
LIN {X 0,Y 197.571,Z 466.888,A -85,B 0,C 180,E1 -21710.834,E2 -21710.834} C_VEL
LIN {X 0,Y 201.235,Z 460.587,A -85,B 0,C 180,E1 -21714.224,E2 -21714.224} C_VEL
LIN {X 0,Y 204.722,Z 453.768,A -85,B 0,C 180,E1 -21717.053,E2 -21717.053} C_VEL
LIN {X 0,Y 208.915,Z 445.253,A -85,B 0,C 180,E1 -21719.745,E2 -21719.745} C_VEL
LIN {X 0,Y 212.755,Z 436.553,A -85,B 0,C 180,E1 -21721.903,E2 -21721.903} C_VEL
LIN {X 0,Y 216.863,Z 425.89,A -85,B 0,C 180,E1 -21723.985,E2 -21723.985} C_VEL
LIN {X 0,Y 220.469,Z 415.229,A -85,B 0,C 180,E1 -21725.571,E2 -21725.571} C_VEL
LIN {X 0,Y 223.725,Z 403.344,A -85,B 0,C 180,E1 -21726.922,E2 -21726.922} C_VEL
LIN {X 0,Y 226.393,Z 391.028,A -85,B 0,C 180,E1 -21727.951,E2 -21727.951} C_VEL
LIN {X 0,Y 228.374,Z 378.254,A -85,B 0,C 180,E1 -21728.69,E2 -21728.69} C_VEL
LIN {X 0,Y 229.751,Z 362.373,A -85,B 0,C 180,E1 -21729.233,E2 -21729.233} C_VEL
LIN {X 0,Y 231.742,Z 328.597,A -85,B 0,C 180,E1 -21730.275,E2 -21730.275} C_VEL
LIN {X 0,Y 226.384,Z 316.303,A -85,B 0,C 180,E1 -21732.406,E2 -21732.406} C_VEL
LIN {X 0,Y 221.669,Z 306.779,A -85,B 0,C 180,E1 -21734.388,E2 -21734.388} C_VEL
LIN {X 0,Y 216.043,Z 297.065,A -85,B 0,C 180,E1 -21736.903,E2 -21736.903} C_VEL
LIN {X 0,Y 212.284,Z 291.017,A -85,B 0,C 180,E1 -21738.766,E2 -21738.766} C_VEL
LIN {X 0,Y 209.849,Z 287.347,A -85,B 0,C 180,E1 -21740.045,E2 -21740.045} C_VEL
LIN {X 0,Y 206.545,Z 282.487,A -85,B 0,C 180,E1 -21741.901,E2 -21741.901} C_VEL
LIN {X 0,Y 202.234,Z 276.441,A -85,B 0,C 180,E1 -21744.587,E2 -21744.587} C_VEL
LIN {X 0,Y 199.525,Z 272.95,A -85,B 0,C 180,E1 -21746.49,E2 -21746.49} C_VEL
LIN {X 0,Y 198.063,Z 270.929,A -85,B 0,C 180,E1 -21747.615,E2 -21747.615} C_VEL
LIN {X 0,Y 193.262,Z 265.19,A -85,B 0,C 180,E1 -21751.853,E2 -21751.853} C_VEL
LIN {X 0,Y 192.819,Z 264.107,A -85,B 0,C 180,E1 -21752.888,E2 -21752.888} C_VEL
LIN {X 0,Y 192.585,Z 263.012,A -85,B 0,C 180,E1 -21754.898,E2 -21754.898} C_VEL
LIN {X 0,Y 192.576,Z 262.983,A -85,B 0,C 180,E1 -21758.588,E2 -21758.588} C_VEL
LIN {X 0,Y 192.711,Z 262.965,A -85,B 0,C 180,E1 -21763.029,E2 -21763.029} C_VEL
LIN {X 0,Y 192.784,Z 262.956,A -85,B 0,C 180,E1 -21767.358,E2 -21767.358} C_VEL
LIN {X 0,Y 193.016,Z 262.928,A -85,B 0,C 180,E1 -21771.617,E2 -21771.617} C_VEL
LIN {X 0,Y 193.216,Z 262.905,A -85,B 0,C 180,E1 -21777.907,E2 -21777.907} C_VEL
LIN {X 0,Y 193.4,Z 262.886,A -85,B 0,C 180,E1 -21779.992,E2 -21779.992} C_VEL
LIN {X 0,Y 192.922,Z 262.947,A -85,B 0,C 180,E1 -21784.17,E2 -21784.17} C_VEL
LIN {X 0,Y 192.975,Z 263.079,A -85,B 0,C 180,E1 -21786.789,E2 -21786.789} C_VEL
LIN {X 0,Y 194.184,Z 266.081,A -85,B 0,C 180,E1 -21788.316,E2 -21788.316} C_VEL
LIN {X 0,Y 196.218,Z 268.066,A -85,B 0,C 180,E1 -21790.068,E2 -21790.068} C_VEL
LIN {X 0,Y 197.701,Z 269.043,A -85,B 0,C 180,E1 -21791.202,E2 -21791.202} C_VEL
LIN {X 0,Y 199.389,Z 272.139,A -85,B 0,C 180,E1 -21792.589,E2 -21792.589} C_VEL
LIN {X 0,Y 202.199,Z 274.74,A -85,B 0,C 180,E1 -21794.49,E2 -21794.49} C_VEL
LIN {X 0,Y 204.573,Z 278.196,A -85,B 0,C 180,E1 -21796.041,E2 -21796.041} C_VEL
LIN {X 0,Y 207.027,Z 281.156,A -85,B 0,C 180,E1 -21797.474,E2 -21797.474} C_VEL
LIN {X 0,Y 211.129,Z 287.005,A -85,B 0,C 180,E1 -21799.725,E2 -21799.725} C_VEL
LIN {X 0,Y 215.163,Z 293.074,A -85,B 0,C 180,E1 -21801.755,E2 -21801.755} C_VEL
LIN {X 0,Y 219.357,Z 299.939,A -85,B 0,C 180,E1 -21803.691,E2 -21803.691} C_VEL
LIN {X 0,Y 225.504,Z 311.062,A -85,B 0,C 180,E1 -21806.295,E2 -21806.295} C_VEL
LIN {X 0,Y 230.883,Z 322.436,A -85,B 0,C 180,E1 -21808.434,E2 -21808.434} C_VEL
LIN {X 0,Y 231.979,Z 325.079,A -85,B 0,C 180,E1 -21808.863,E2 -21808.863} C_VEL
LIN {X 0,Y 228.966,Z 370.282,A -85,B 0,C 180,E1 -21810.246,E2 -21810.246} C_VEL
LIN {X 0,Y 227.088,Z 384.163,A -85,B 0,C 180,E1 -21810.984,E2 -21810.984} C_VEL
LIN {X 0,Y 224.662,Z 396.399,A -85,B 0,C 180,E1 -21811.953,E2 -21811.953} C_VEL
LIN {X 0,Y 221.644,Z 408.222,A -85,B 0,C 180,E1 -21813.253,E2 -21813.253} C_VEL
LIN {X 0,Y 218.265,Z 419.064,A -85,B 0,C 180,E1 -21814.812,E2 -21814.812} C_VEL
LIN {X 0,Y 214.568,Z 429.055,A -85,B 0,C 180,E1 -21816.638,E2 -21816.638} C_VEL
LIN {X 0,Y 210.25,Z 439.084,A -85,B 0,C 180,E1 -21819.003,E2 -21819.003} C_VEL
LIN {X 0,Y 206.326,Z 447.218,A -85,B 0,C 180,E1 -21821.469,E2 -21821.469} C_VEL
LIN {X 0,Y 202.611,Z 454.319,A -85,B 0,C 180,E1 -21824.225,E2 -21824.225} C_VEL
LIN {X 0,Y 199.778,Z 459.322,A -85,B 0,C 180,E1 -21826.691,E2 -21826.691} C_VEL
LIN {X 0,Y 196.651,Z 464.487,A -85,B 0,C 180,E1 -21829.967,E2 -21829.967} C_VEL
LIN {X 0,Y 194.671,Z 467.55,A -85,B 0,C 180,E1 -21832.567,E2 -21832.567} C_VEL
LIN {X 0,Y 193.52,Z 469.316,A -85,B 0,C 180,E1 -21834.479,E2 -21834.479} C_VEL
LIN {X 0,Y 192.105,Z 471.233,A -85,B 0,C 180,E1 -21837.274,E2 -21837.274} C_VEL
